C03601=1040.712,-116.263,-73.766,168.679,35.382,156.678
C03602=1040.719,-115.977,-73.778,168.682,35.382,156.678
C03603=1040.726,-115.691,-73.788,168.684,35.381,156.678
C03604=1040.733,-115.404,-73.799,168.687,35.381,156.678
C03605=1040.739,-115.155,-73.808,168.690,35.381,156.678
C03606=1040.745,-114.905,-73.817,168.692,35.380,156.678
C03607=1040.751,-114.656,-73.827,168.695,35.380,156.678
C03608=1040.757,-114.406,-73.837,168.698,35.380,156.678
C03609=1040.763,-114.156,-73.846,168.700,35.379,156.678
C03610=1040.769,-113.906,-73.855,168.703,35.378,156.677
C03611=1040.775,-113.656,-73.865,168.705,35.379,156.677
C03612=1040.781,-113.406,-73.874,168.708,35.378,156.677
C03613=1040.787,-113.157,-73.883,168.710,35.378,156.677
C03614=1040.793,-112.907,-73.893,168.712,35.377,156.677
C03615=1040.799,-112.657,-73.902,168.714,35.377,156.677
C03616=1040.806,-112.407,-73.912,168.717,35.377,156.677
C03617=1040.812,-112.158,-73.922,168.719,35.376,156.677
C03618=1040.818,-111.908,-73.931,168.722,35.376,156.677
C03619=1040.823,-111.658,-73.941,168.724,35.376,156.677
C03620=1040.829,-111.408,-73.951,168.727,35.375,156.677
C03621=1040.836,-111.158,-73.960,168.729,35.375,156.677
C03622=1040.841,-110.909,-73.970,168.732,35.375,156.676
C03623=1040.847,-110.659,-73.979,168.734,35.375,156.676
C03624=1040.854,-110.409,-73.989,168.737,35.374,156.676
C03625=1040.860,-110.160,-73.999,168.740,35.374,156.676
C03626=1040.866,-109.911,-74.009,168.742,35.374,156.676
C03627=1040.872,-109.661,-74.018,168.745,35.373,156.676
C03628=1040.879,-109.411,-74.028,168.747,35.373,156.676
C03629=1040.885,-109.161,-74.037,168.750,35.373,156.676
C03630=1040.891,-108.911,-74.047,168.752,35.373,156.676
C03631=1040.897,-108.662,-74.056,168.755,35.372,156.676
C03632=1040.903,-108.412,-74.066,168.757,35.372,156.676
C03633=1040.909,-108.162,-74.076,168.760,35.372,156.676
C03634=1040.915,-107.912,-74.086,168.762,35.372,156.676
C03635=1040.921,-107.663,-74.096,168.765,35.371,156.675
C03636=1040.927,-107.413,-74.106,168.767,35.371,156.675
C03637=1040.934,-107.163,-74.115,168.770,35.371,156.675
C03638=1040.940,-106.913,-74.125,168.772,35.371,156.675
C03639=1040.945,-106.663,-74.135,168.775,35.370,156.675
C03640=1040.952,-106.414,-74.145,168.777,35.370,156.675
C03641=1040.958,-106.164,-74.155,168.779,35.370,156.675
C03642=1040.964,-105.914,-74.164,168.781,35.370,156.675
C03643=1040.970,-105.665,-74.174,168.784,35.370,156.675
C03644=1040.976,-105.414,-74.184,168.786,35.369,156.675
C03645=1040.982,-105.165,-74.194,168.789,35.369,156.675
C03646=1040.988,-104.915,-74.204,168.791,35.369,156.675
C03647=1040.994,-104.666,-74.213,168.794,35.369,156.675
C03648=1041.000,-104.416,-74.224,168.796,35.369,156.675
C03649=1041.006,-104.166,-74.234,168.799,35.368,156.674
C03650=1041.013,-103.917,-74.243,168.801,35.368,156.674
C03651=1041.019,-103.667,-74.253,168.804,35.368,156.674
C03652=1041.024,-103.417,-74.264,168.806,35.368,156.674
C03653=1041.031,-103.168,-74.273,168.809,35.368,156.674
C03654=1041.037,-102.918,-74.283,168.811,35.367,156.674
C03655=1041.043,-102.668,-74.294,168.814,35.368,156.674
C03656=1041.049,-102.418,-74.303,168.816,35.368,156.674
C03657=1041.055,-102.169,-74.313,168.819,35.367,156.674
C03658=1041.061,-101.919,-74.323,168.821,35.367,156.674
C03659=1041.067,-101.669,-74.334,168.824,35.367,156.674
C03660=1041.074,-101.419,-74.344,168.826,35.367,156.674
C03661=1041.080,-101.170,-74.354,168.829,35.367,156.674
C03662=1041.086,-100.920,-74.364,168.831,35.367,156.674
C03663=1041.092,-100.670,-74.374,168.834,35.366,156.674
C03664=1041.098,-100.421,-74.384,168.836,35.366,156.674
C03665=1041.105,-100.134,-74.396,168.839,35.366,156.674
C03666=1041.112,-99.846,-74.408,168.842,35.366,156.673
C03667=1041.120,-99.559,-74.419,168.845,35.366,156.673
C03668=1041.127,-99.272,-74.431,168.847,35.366,156.673
C03669=1041.133,-99.022,-74.441,168.850,35.365,156.673
C03670=1041.139,-98.772,-74.450,168.852,35.365,156.673
C03671=1041.145,-98.523,-74.461,168.855,35.366,156.673
C03672=1041.151,-98.273,-74.471,168.857,35.366,156.673
C03673=1041.157,-98.024,-74.481,168.860,35.365,156.673
C03674=1041.163,-97.773,-74.492,168.862,35.365,156.673
C03675=1041.170,-97.524,-74.502,168.865,35.365,156.673
C03676=1041.175,-97.274,-74.512,168.867,35.365,156.673
C03677=1041.182,-97.025,-74.522,168.870,35.365,156.673
C03678=1041.187,-96.775,-74.533,168.871,35.365,156.673
C03679=1041.194,-96.525,-74.543,168.874,35.365,156.673
C03680=1041.199,-96.276,-74.554,168.876,35.365,156.673
C03681=1041.206,-96.025,-74.564,168.878,35.365,156.673
C03682=1041.212,-95.776,-74.575,168.881,35.365,156.673
C03683=1041.218,-95.526,-74.585,168.883,35.365,156.673
C03684=1041.224,-95.277,-74.595,168.886,35.365,156.673
C03685=1041.230,-95.027,-74.606,168.888,35.365,156.673
C03686=1041.236,-94.778,-74.616,168.891,35.365,156.673
C03687=1041.242,-94.527,-74.627,168.893,35.365,156.673
C03688=1041.248,-94.278,-74.637,168.895,35.365,156.673
C03689=1041.254,-94.028,-74.648,168.898,35.366,156.673
C03690=1041.260,-93.778,-74.658,168.900,35.365,156.673
C03691=1041.266,-93.529,-74.668,168.903,35.365,156.673
C03692=1041.272,-93.279,-74.680,168.905,35.365,156.673
C03693=1041.279,-93.029,-74.689,168.908,35.365,156.673
C03694=1041.284,-92.780,-74.700,168.910,35.365,156.673
C03695=1041.290,-92.530,-74.711,168.913,35.365,156.673
C03696=1041.297,-92.280,-74.721,168.915,35.365,156.672
C03697=1041.303,-92.030,-74.732,168.917,35.366,156.672
C03698=1041.309,-91.781,-74.742,168.920,35.366,156.672
C03699=1041.315,-91.531,-74.753,168.922,35.366,156.672
C03700=1041.321,-91.281,-74.764,168.925,35.366,156.672
C03701=1041.327,-91.031,-74.774,168.927,35.366,156.672
C03702=1041.333,-90.782,-74.785,168.930,35.366,156.672
C03703=1041.340,-90.533,-74.795,168.932,35.366,156.672
C03704=1041.346,-90.283,-74.806,168.934,35.366,156.672
C03705=1041.351,-90.033,-74.816,168.937,35.366,156.672
C03706=1041.358,-89.783,-74.826,168.939,35.366,156.672
C03707=1041.364,-89.533,-74.838,168.942,35.366,156.672
C03708=1041.370,-89.284,-74.849,168.944,35.366,156.672
C03709=1041.376,-89.034,-74.859,168.946,35.366,156.672
C03710=1041.382,-88.785,-74.870,168.949,35.366,156.672
C03711=1041.389,-88.535,-74.880,168.951,35.367,156.672
C03712=1041.395,-88.285,-74.891,168.954,35.367,156.672
C03713=1041.400,-88.036,-74.901,168.956,35.367,156.672
C03714=1041.407,-87.786,-74.912,168.959,35.367,156.672
C03715=1041.413,-87.536,-74.923,168.961,35.367,156.672
C03716=1041.419,-87.287,-74.934,168.963,35.367,156.672
C03717=1041.426,-87.037,-74.944,168.966,35.367,156.672
C03718=1041.432,-86.787,-74.955,168.968,35.367,156.672
C03719=1041.438,-86.537,-74.967,168.971,35.367,156.672
C03720=1041.445,-86.288,-74.977,168.973,35.367,156.672
C03721=1041.450,-86.038,-74.988,168.975,35.367,156.672
C03722=1041.456,-85.788,-74.998,168.978,35.367,156.672
C03723=1041.463,-85.538,-75.009,168.980,35.367,156.672
C03724=1041.469,-85.289,-75.019,168.983,35.367,156.672
C03725=1041.475,-85.039,-75.031,168.985,35.368,156.672
C03726=1041.481,-84.790,-75.041,168.988,35.368,156.672
C03727=1041.488,-84.539,-75.052,168.990,35.368,156.672
C03728=1041.493,-84.290,-75.063,168.992,35.368,156.672
C03729=1041.501,-84.005,-75.076,168.995,35.369,156.672
C03730=1041.508,-83.721,-75.088,168.998,35.369,156.672
C03731=1041.515,-83.435,-75.100,169.001,35.369,156.672
C03732=1041.522,-83.151,-75.113,169.003,35.369,156.672
C03733=1041.529,-82.901,-75.124,169.006,35.369,156.672
C03734=1041.535,-82.652,-75.135,169.008,35.369,156.672
C03735=1041.541,-82.402,-75.146,169.011,35.369,156.672
C03736=1041.547,-82.152,-75.157,169.013,35.369,156.672
C03737=1041.554,-81.902,-75.167,169.015,35.369,156.672
C03738=1041.560,-81.653,-75.178,169.018,35.369,156.672
C03739=1041.566,-81.403,-75.189,169.020,35.370,156.672
C03740=1041.573,-81.153,-75.200,169.023,35.370,156.672
C03741=1041.579,-80.903,-75.211,169.025,35.370,156.672
C03742=1041.585,-80.654,-75.222,169.027,35.370,156.672
C03743=1041.591,-80.403,-75.233,169.030,35.370,156.672
C03744=1041.598,-80.155,-75.244,169.032,35.370,156.672
C03745=1041.604,-79.905,-75.255,169.035,35.370,156.672
C03746=1041.610,-79.655,-75.266,169.037,35.370,156.672
C03747=1041.616,-79.405,-75.277,169.039,35.371,156.672
C03748=1041.622,-79.156,-75.288,169.042,35.371,156.672
C03749=1041.628,-78.905,-75.300,169.044,35.371,156.672
C03750=1041.634,-78.656,-75.311,169.046,35.372,156.672
C03751=1041.642,-78.407,-75.322,169.049,35.372,156.672
C03752=1041.647,-78.157,-75.333,169.051,35.372,156.672
C03753=1041.654,-77.907,-75.344,169.053,35.372,156.672
C03754=1041.660,-77.658,-75.356,169.056,35.373,156.672
C03755=1041.666,-77.408,-75.367,169.058,35.373,156.672
C03756=1041.672,-77.158,-75.378,169.060,35.373,156.672
C03757=1041.678,-76.909,-75.390,169.063,35.374,156.672
C03758=1041.684,-76.659,-75.400,169.065,35.374,156.672
C03759=1041.690,-76.409,-75.412,169.068,35.374,156.672
C03760=1041.696,-76.160,-75.423,169.070,35.375,156.672
C03761=1041.703,-75.910,-75.435,169.072,35.375,156.672
C03762=1041.709,-75.661,-75.445,169.075,35.375,156.672
C03763=1041.715,-75.410,-75.457,169.077,35.375,156.672
C03764=1041.722,-75.161,-75.469,169.079,35.376,156.672
C03765=1041.727,-74.911,-75.480,169.082,35.376,156.672
C03766=1041.734,-74.661,-75.491,169.084,35.376,156.672
C03767=1041.740,-74.412,-75.502,169.086,35.376,156.672
C03768=1041.746,-74.162,-75.514,169.089,35.376,156.672
C03769=1041.752,-73.913,-75.525,169.091,35.377,156.672
C03770=1041.758,-73.663,-75.536,169.093,35.377,156.672
C03771=1041.765,-73.413,-75.548,169.096,35.378,156.672
C03772=1041.771,-73.164,-75.559,169.098,35.378,156.672
C03773=1041.776,-72.913,-75.571,169.100,35.379,156.673
C03774=1041.782,-72.665,-75.583,169.103,35.379,156.672
C03775=1041.789,-72.414,-75.594,169.105,35.380,156.673
C03776=1041.795,-72.166,-75.606,169.107,35.380,156.673
C03777=1041.800,-71.915,-75.617,169.109,35.380,156.673
C03778=1041.807,-71.665,-75.629,169.112,35.380,156.673
C03779=1041.813,-71.416,-75.640,169.114,35.381,156.673
C03780=1041.820,-71.166,-75.652,169.116,35.381,156.673
C03781=1041.825,-70.917,-75.664,169.119,35.382,156.673
C03782=1041.831,-70.667,-75.676,169.121,35.382,156.673
C03783=1041.837,-70.417,-75.687,169.123,35.383,156.673
C03784=1041.844,-70.168,-75.698,169.126,35.383,156.673
C03785=1041.850,-69.918,-75.710,169.128,35.383,156.673
C03786=1041.855,-69.669,-75.722,169.130,35.384,156.673
C03787=1041.862,-69.419,-75.734,169.132,35.384,156.673
C03788=1041.868,-69.169,-75.745,169.135,35.385,156.673
C03789=1041.874,-68.920,-75.757,169.137,35.385,156.673
C03790=1041.880,-68.669,-75.768,169.139,35.386,156.673
C03791=1041.886,-68.420,-75.780,169.142,35.386,156.673
C03792=1041.893,-68.171,-75.792,169.144,35.386,156.673
C03793=1041.899,-67.888,-75.805,169.147,35.387,156.673
C03794=1041.907,-67.605,-75.818,169.149,35.387,156.673
C03795=1041.914,-67.323,-75.832,169.152,35.388,156.673
C03796=1041.920,-67.040,-75.845,169.154,35.389,156.674
C03797=1041.926,-66.790,-75.857,169.157,35.389,156.674
C03798=1041.933,-66.540,-75.869,169.159,35.390,156.674
C03799=1041.939,-66.291,-75.881,169.161,35.390,156.674
C03800=1041.945,-66.042,-75.892,169.163,35.390,156.674
C03801=1041.951,-65.791,-75.904,169.166,35.390,156.674
C03802=1041.957,-65.542,-75.916,169.168,35.391,156.674
C03803=1041.964,-65.293,-75.928,169.170,35.392,156.674
C03804=1041.969,-65.042,-75.940,169.173,35.392,156.674
C03805=1041.976,-64.793,-75.952,169.175,35.393,156.674
C03806=1041.982,-64.544,-75.963,169.177,35.393,156.674
C03807=1041.989,-64.294,-75.975,169.179,35.393,156.674
C03808=1041.994,-64.044,-75.987,169.182,35.394,156.674
C03809=1042.001,-63.794,-75.999,169.184,35.394,156.674
C03810=1042.007,-63.545,-76.011,169.186,35.395,156.674
C03811=1042.013,-63.295,-76.023,169.189,35.395,156.674
C03812=1042.019,-63.045,-76.034,169.192,35.396,156.674
C03813=1042.026,-62.796,-76.046,169.194,35.396,156.674
C03814=1042.031,-62.546,-76.059,169.196,35.396,156.674
C03815=1042.038,-62.297,-76.071,169.199,35.397,156.675
C03816=1042.044,-62.047,-76.082,169.201,35.398,156.675
C03817=1042.050,-61.797,-76.095,169.203,35.398,156.675
C03818=1042.057,-61.547,-76.106,169.205,35.399,156.675
C03819=1042.063,-61.298,-76.118,169.208,35.399,156.675
C03820=1042.069,-61.049,-76.130,169.210,35.399,156.675
C03821=1042.075,-60.799,-76.142,169.212,35.400,156.675
C03822=1042.082,-60.549,-76.154,169.214,35.400,156.675
C03823=1042.088,-60.300,-76.166,169.217,35.401,156.675
C03824=1042.094,-60.050,-76.179,169.219,35.402,156.675
C03825=1042.100,-59.800,-76.190,169.221,35.402,156.675
C03826=1042.107,-59.551,-76.202,169.224,35.402,156.675
C03827=1042.113,-59.301,-76.214,169.226,35.403,156.675
C03828=1042.119,-59.051,-76.226,169.228,35.403,156.675
C03829=1042.126,-58.802,-76.238,169.230,35.404,156.675
C03830=1042.132,-58.552,-76.251,169.233,35.405,156.675
C03831=1042.139,-58.302,-76.263,169.235,35.405,156.675
C03832=1042.144,-58.053,-76.275,169.237,35.405,156.675
C03833=1042.150,-57.804,-76.287,169.239,35.406,156.676
C03834=1042.157,-57.554,-76.299,169.242,35.406,156.676
C03835=1042.163,-57.304,-76.311,169.244,35.407,156.676
C03836=1042.170,-57.055,-76.323,169.246,35.407,156.676
C03837=1042.176,-56.805,-76.335,169.248,35.408,156.676
C03838=1042.182,-56.555,-76.348,169.251,35.408,156.676
C03839=1042.189,-56.306,-76.360,169.253,35.409,156.676
C03840=1042.196,-56.056,-76.372,169.255,35.409,156.676
C03841=1042.201,-55.806,-76.384,169.257,35.410,156.676
C03842=1042.208,-55.556,-76.396,169.260,35.410,156.676
C03843=1042.214,-55.308,-76.408,169.262,35.410,156.676
C03844=1042.220,-55.058,-76.420,169.264,35.411,156.676
C03845=1042.227,-54.808,-76.432,169.266,35.412,156.676
C03846=1042.233,-54.558,-76.445,169.269,35.412,156.676
C03847=1042.239,-54.309,-76.457,169.271,35.413,156.676
C03848=1042.246,-54.059,-76.469,169.273,35.413,156.676
C03849=1042.252,-53.809,-76.481,169.275,35.414,156.677
C03850=1042.259,-53.560,-76.494,169.278,35.414,156.677
C03851=1042.265,-53.310,-76.507,169.280,35.415,156.677
C03852=1042.271,-53.061,-76.519,169.282,35.416,156.677
C03853=1042.278,-52.811,-76.531,169.284,35.416,156.677
C03854=1042.284,-52.561,-76.543,169.286,35.416,156.677
C03855=1042.291,-52.312,-76.555,169.289,35.417,156.677
C03856=1042.296,-52.062,-76.568,169.291,35.417,156.677
C03857=1042.305,-51.781,-76.581,169.293,35.418,156.677
C03858=1042.312,-51.499,-76.596,169.297,35.419,156.677
C03859=1042.318,-51.218,-76.609,169.299,35.419,156.677
C03860=1042.326,-50.937,-76.624,169.302,35.420,156.677
C03861=1042.332,-50.687,-76.636,169.304,35.420,156.677
C03862=1042.338,-50.437,-76.648,169.306,35.421,156.677
C03863=1042.345,-50.188,-76.660,169.309,35.421,156.677
C03864=1042.351,-49.938,-76.673,169.311,35.422,156.678
C03865=1042.357,-49.688,-76.686,169.313,35.423,156.678
C03866=1042.364,-49.439,-76.698,169.315,35.424,156.678
C03867=1042.370,-49.189,-76.710,169.317,35.424,156.678
C03868=1042.376,-48.940,-76.724,169.319,35.425,156.678
C03869=1042.382,-48.690,-76.736,169.322,35.426,156.678
C03870=1042.388,-48.440,-76.748,169.324,35.426,156.678
C03871=1042.395,-48.191,-76.761,169.326,35.427,156.678
C03872=1042.400,-47.941,-76.774,169.328,35.428,156.678
C03873=1042.407,-47.692,-76.787,169.330,35.428,156.678
C03874=1042.413,-47.442,-76.799,169.333,35.429,156.679
C03875=1042.419,-47.192,-76.812,169.335,35.430,156.679
C03876=1042.425,-46.943,-76.825,169.337,35.431,156.679
C03877=1042.431,-46.693,-76.838,169.339,35.431,156.679
C03878=1042.438,-46.444,-76.850,169.341,35.432,156.679
C03879=1042.445,-46.194,-76.863,169.343,35.433,156.679
C03880=1042.451,-45.944,-76.876,169.346,35.433,156.679
C03881=1042.457,-45.695,-76.889,169.348,35.434,156.679
C03882=1042.463,-45.445,-76.902,169.350,35.435,156.679
C03883=1042.469,-45.195,-76.914,169.352,35.435,156.679
C03884=1042.476,-44.946,-76.927,169.354,35.436,156.679
C03885=1042.482,-44.696,-76.939,169.356,35.436,156.680
C03886=1042.488,-44.447,-76.953,169.359,35.437,156.680
C03887=1042.494,-44.197,-76.965,169.362,35.438,156.680
C03888=1042.501,-43.948,-76.978,169.364,35.438,156.680
C03889=1042.507,-43.698,-76.990,169.366,35.439,156.680
C03890=1042.513,-43.449,-77.004,169.368,35.440,156.680
C03891=1042.519,-43.198,-77.017,169.370,35.440,156.680
C03892=1042.526,-42.949,-77.029,169.372,35.441,156.680
C03893=1042.532,-42.699,-77.042,169.375,35.442,156.680
C03894=1042.538,-42.450,-77.055,169.377,35.443,156.680
C03895=1042.544,-42.200,-77.068,169.379,35.443,156.681
C03896=1042.551,-41.951,-77.080,169.381,35.444,156.681
C03897=1042.557,-41.701,-77.093,169.383,35.445,156.681
C03898=1042.564,-41.451,-77.107,169.385,35.445,156.681
C03899=1042.570,-41.202,-77.120,169.387,35.446,156.681
C03900=1042.576,-40.952,-77.132,169.390,35.447,156.681
C03901=1042.582,-40.703,-77.146,169.392,35.447,156.681
C03902=1042.589,-40.453,-77.158,169.394,35.448,156.681
C03903=1042.595,-40.204,-77.171,169.396,35.449,156.681
C03904=1042.602,-39.954,-77.185,169.398,35.450,156.682
C03905=1042.608,-39.704,-77.197,169.400,35.451,156.682
C03906=1042.614,-39.455,-77.210,169.402,35.452,156.682
C03907=1042.621,-39.205,-77.222,169.405,35.452,156.682
C03908=1042.627,-38.956,-77.236,169.407,35.453,156.682
C03909=1042.634,-38.706,-77.249,169.409,35.454,156.682
C03910=1042.640,-38.456,-77.262,169.411,35.454,156.682
C03911=1042.646,-38.207,-77.275,169.414,35.455,156.682
C03912=1042.652,-37.958,-77.288,169.416,35.456,156.682
C03913=1042.658,-37.708,-77.301,169.418,35.456,156.682
C03914=1042.665,-37.458,-77.314,169.420,35.458,156.683
C03915=1042.671,-37.209,-77.328,169.423,35.459,156.683
C03916=1042.677,-36.959,-77.341,169.425,35.459,156.683
C03917=1042.683,-36.710,-77.354,169.427,35.460,156.683
C03918=1042.689,-36.460,-77.367,169.429,35.461,156.683
C03919=1042.695,-36.210,-77.381,169.431,35.461,156.683
C03920=1042.702,-35.961,-77.394,169.433,35.463,156.683
C03921=1042.708,-35.680,-77.408,169.435,35.463,156.683
C03922=1042.716,-35.399,-77.424,169.438,35.464,156.684
C03923=1042.723,-35.118,-77.439,169.440,35.465,156.684
C03924=1042.730,-34.837,-77.453,169.442,35.466,156.684
C03925=1042.737,-34.587,-77.467,169.445,35.467,156.684
C03926=1042.743,-34.338,-77.480,169.447,35.467,156.684
C03927=1042.749,-34.088,-77.493,169.449,35.469,156.684
C03928=1042.755,-33.839,-77.506,169.451,35.469,156.684
C03929=1042.762,-33.589,-77.520,169.453,35.470,156.684
C03930=1042.767,-33.340,-77.534,169.455,35.471,156.685
C03931=1042.773,-33.090,-77.547,169.458,35.472,156.685
C03932=1042.780,-32.840,-77.560,169.460,35.473,156.685
C03933=1042.786,-32.591,-77.574,169.462,35.474,156.685
C03934=1042.792,-32.341,-77.586,169.464,35.474,156.685
C03935=1042.799,-32.092,-77.600,169.466,35.475,156.685
C03936=1042.805,-31.842,-77.613,169.469,35.476,156.685
C03937=1042.812,-31.593,-77.626,169.471,35.477,156.686
C03938=1042.818,-31.343,-77.640,169.473,35.478,156.686
C03939=1042.825,-31.093,-77.653,169.475,35.478,156.686
C03940=1042.831,-30.844,-77.667,169.477,35.479,156.686
C03941=1042.836,-30.595,-77.681,169.479,35.480,156.686
C03942=1042.843,-30.345,-77.694,169.481,35.481,156.686
C03943=1042.849,-30.095,-77.707,169.483,35.482,156.686
C03944=1042.856,-29.846,-77.721,169.485,35.483,156.686
C03945=1042.862,-29.596,-77.734,169.487,35.483,156.686
C03946=1042.869,-29.347,-77.748,169.489,35.484,156.687
C03947=1042.875,-29.098,-77.761,169.491,35.485,156.687
C03948=1042.882,-28.848,-77.775,169.493,35.486,156.687
C03949=1042.888,-28.598,-77.788,169.495,35.487,156.687
C03950=1042.894,-28.348,-77.802,169.498,35.487,156.687
C03951=1042.900,-28.099,-77.815,169.501,35.489,156.687
C03952=1042.906,-27.850,-77.829,169.503,35.489,156.687
C03953=1042.913,-27.600,-77.842,169.505,35.490,156.687
C03954=1042.919,-27.350,-77.855,169.507,35.491,156.688
C03955=1042.926,-27.100,-77.869,169.509,35.491,156.688
C03956=1042.932,-26.851,-77.882,169.511,35.493,156.688
C03957=1042.938,-26.602,-77.896,169.513,35.493,156.688
C03958=1042.945,-26.352,-77.910,169.515,35.494,156.688
C03959=1042.951,-26.102,-77.923,169.517,35.495,156.688
C03960=1042.957,-25.853,-77.938,169.519,35.496,156.688
C03961=1042.964,-25.603,-77.951,169.521,35.497,156.689
C03962=1042.969,-25.354,-77.965,169.523,35.498,156.689
C03963=1042.976,-25.104,-77.979,169.525,35.499,156.689
C03964=1042.982,-24.855,-77.992,169.527,35.500,156.689
C03965=1042.988,-24.605,-78.006,169.529,35.501,156.689
C03966=1042.995,-24.356,-78.020,169.531,35.502,156.689
C03967=1043.001,-24.106,-78.034,169.533,35.503,156.689
C03968=1043.007,-23.856,-78.048,169.536,35.504,156.690
C03969=1043.013,-23.607,-78.061,169.538,35.505,156.690
C03970=1043.019,-23.358,-78.074,169.540,35.506,156.690
C03971=1043.026,-23.108,-78.089,169.542,35.506,156.690
C03972=1043.032,-22.859,-78.103,169.544,35.508,156.690
C03973=1043.038,-22.608,-78.117,169.546,35.508,156.690
C03974=1043.044,-22.359,-78.130,169.548,35.510,156.691
C03975=1043.051,-22.110,-78.144,169.550,35.510,156.691
C03976=1043.057,-21.860,-78.158,169.552,35.511,156.691
C03977=1043.064,-21.610,-78.172,169.554,35.512,156.691
C03978=1043.069,-21.361,-78.186,169.556,35.513,156.691
C03979=1043.076,-21.112,-78.200,169.558,35.514,156.691
C03980=1043.082,-20.862,-78.213,169.560,35.515,156.691
C03981=1043.088,-20.612,-78.227,169.562,35.516,156.691
C03982=1043.095,-20.363,-78.242,169.564,35.517,156.692
C03983=1043.101,-20.114,-78.255,169.566,35.518,156.692
C03984=1043.107,-19.864,-78.269,169.569,35.519,156.692
C03985=1043.115,-19.582,-78.285,169.572,35.520,156.692
C03986=1043.122,-19.301,-78.301,169.574,35.521,156.692
C03987=1043.129,-19.018,-78.316,169.576,35.522,156.692
C03988=1043.136,-18.737,-78.332,169.579,35.523,156.693
C03989=1043.142,-18.487,-78.346,169.581,35.524,156.693
C03990=1043.149,-18.238,-78.360,169.583,35.525,156.693
C03991=1043.155,-17.988,-78.374,169.585,35.526,156.693
C03992=1043.162,-17.739,-78.389,169.586,35.527,156.693
C03993=1043.168,-17.489,-78.402,169.588,35.528,156.693
C03994=1043.174,-17.239,-78.416,169.590,35.529,156.693
C03995=1043.181,-16.990,-78.430,169.592,35.530,156.694
C03996=1043.187,-16.740,-78.444,169.594,35.531,156.694
C03997=1043.193,-16.491,-78.459,169.596,35.531,156.694
C03998=1043.200,-16.241,-78.472,169.598,35.533,156.694
C03999=1043.206,-15.993,-78.487,169.600,35.533,156.694
C04000=1043.213,-15.743,-78.500,169.603,35.535,156.694
C04001=1043.219,-15.492,-78.515,169.605,35.535,156.695
C04002=1043.225,-15.244,-78.529,169.607,35.536,156.695
C04003=1043.231,-14.993,-78.543,169.609,35.537,156.695
C04004=1043.238,-14.745,-78.557,169.611,35.539,156.695
C04005=1043.244,-14.495,-78.572,169.613,35.539,156.695
C04006=1043.250,-14.245,-78.586,169.615,35.541,156.695
C04007=1043.257,-13.996,-78.600,169.617,35.541,156.695
C04008=1043.263,-13.746,-78.614,169.619,35.543,156.696
C04009=1043.269,-13.497,-78.629,169.621,35.543,156.696
C04010=1043.275,-13.247,-78.642,169.623,35.545,156.696
C04011=1043.281,-12.998,-78.657,169.625,35.545,156.696
C04012=1043.288,-12.748,-78.672,169.627,35.547,156.696
C04013=1043.294,-12.498,-78.686,169.629,35.548,156.697
C04014=1043.300,-12.249,-78.700,169.631,35.549,156.697
C04015=1043.306,-11.999,-78.714,169.634,35.550,156.697
C04016=1043.313,-11.750,-78.728,169.636,35.551,156.697
C04017=1043.319,-11.501,-78.743,169.638,35.552,156.697
C04018=1043.325,-11.251,-78.758,169.640,35.553,156.697
C04019=1043.332,-11.002,-78.772,169.642,35.554,156.698
C04020=1043.338,-10.752,-78.787,169.644,35.555,156.698
C04021=1043.344,-10.503,-78.800,169.646,35.556,156.698
C04022=1043.351,-10.253,-78.815,169.647,35.557,156.698
C04023=1043.357,-10.004,-78.830,169.649,35.558,156.698
C04024=1043.363,-9.754,-78.844,169.651,35.559,156.698
C04025=1043.369,-9.504,-78.859,169.653,35.560,156.698
C04026=1043.376,-9.255,-78.873,169.655,35.561,156.699
C04027=1043.382,-9.006,-78.887,169.657,35.562,156.699
C04028=1043.388,-8.756,-78.902,169.660,35.563,156.699
C04029=1043.395,-8.507,-78.916,169.662,35.564,156.699
C04030=1043.401,-8.258,-78.931,169.664,35.565,156.699
C04031=1043.407,-8.007,-78.945,169.666,35.567,156.700
C04032=1043.414,-7.758,-78.959,169.668,35.567,156.700
C04033=1043.420,-7.509,-78.974,169.670,35.569,156.700
C04034=1043.426,-7.259,-78.989,169.672,35.569,156.700
C04035=1043.432,-7.009,-79.003,169.674,35.571,156.700
C04036=1043.439,-6.760,-79.017,169.676,35.571,156.700
C04037=1043.445,-6.511,-79.032,169.678,35.573,156.701
C04038=1043.452,-6.261,-79.047,169.679,35.574,156.701
C04039=1043.459,-6.012,-79.061,169.681,35.575,156.701
C04040=1043.464,-5.762,-79.075,169.683,35.576,156.701
C04041=1043.471,-5.513,-79.090,169.685,35.577,156.701
C04042=1043.477,-5.263,-79.105,169.688,35.578,156.701
C04043=1043.484,-5.014,-79.119,169.690,35.579,156.701
C04044=1043.490,-4.765,-79.134,169.692,35.580,156.702
C04045=1043.496,-4.515,-79.149,169.694,35.581,156.702
C04046=1043.502,-4.265,-79.163,169.696,35.582,156.702
C04047=1043.509,-4.015,-79.177,169.698,35.583,156.702
C04048=1043.515,-3.766,-79.192,169.700,35.584,156.702
C04049=1043.523,-3.483,-79.209,169.702,35.585,156.703
C04050=1043.530,-3.199,-79.226,169.704,35.587,156.703
C04051=1043.537,-2.915,-79.243,169.706,35.588,156.703
C04052=1043.544,-2.633,-79.260,169.708,35.589,156.703
C04053=1043.550,-2.384,-79.274,169.710,35.590,156.703
C04054=1043.556,-2.134,-79.289,169.712,35.591,156.704
C04055=1043.563,-1.884,-79.304,169.715,35.592,156.704
C04056=1043.569,-1.635,-79.319,169.717,35.594,156.704
C04057=1043.575,-1.386,-79.334,169.719,35.595,156.704
C04058=1043.581,-1.136,-79.349,169.721,35.596,156.704
C04059=1043.587,-0.886,-79.364,169.722,35.597,156.705
C04060=1043.594,-0.637,-79.379,169.724,35.598,156.705
C04061=1043.600,-0.388,-79.393,169.726,35.600,156.705
C04062=1043.606,-0.138,-79.408,169.728,35.600,156.705
C04063=1043.612,0.111,-79.423,169.730,35.602,156.705
C04064=1043.619,0.361,-79.438,169.732,35.603,156.706
C04065=1043.624,0.610,-79.453,169.734,35.604,156.706
C04066=1043.630,0.860,-79.468,169.736,35.605,156.706
C04067=1043.637,1.110,-79.483,169.738,35.606,156.706
C04068=1043.643,1.359,-79.498,169.740,35.608,156.706
C04069=1043.649,1.609,-79.513,169.742,35.609,156.706
C04070=1043.655,1.858,-79.528,169.744,35.610,156.707
C04071=1043.662,2.107,-79.543,169.746,35.611,156.707
C04072=1043.668,2.357,-79.558,169.748,35.612,156.707
C04073=1043.675,2.606,-79.573,169.750,35.614,156.707
C04074=1043.681,2.856,-79.588,169.751,35.614,156.707
C04075=1043.687,3.106,-79.603,169.753,35.616,156.708
C04076=1043.693,3.355,-79.618,169.755,35.617,156.708
C04077=1043.700,3.604,-79.633,169.757,35.618,156.708
C04078=1043.706,3.853,-79.648,169.760,35.619,156.708
C04079=1043.713,4.103,-79.663,169.762,35.620,156.708
C04080=1043.718,4.353,-79.679,169.764,35.621,156.709
C04081=1043.725,4.603,-79.694,169.765,35.623,156.709
C04082=1043.731,4.852,-79.709,169.767,35.623,156.709
C04083=1043.737,5.101,-79.724,169.769,35.625,156.709
C04084=1043.744,5.350,-79.739,169.771,35.626,156.709
C04085=1043.750,5.600,-79.754,169.773,35.627,156.710
C04086=1043.756,5.850,-79.769,169.775,35.628,156.710
C04087=1043.763,6.099,-79.784,169.777,35.629,156.710
C04088=1043.769,6.348,-79.799,169.778,35.631,156.710
C04089=1043.776,6.598,-79.814,169.780,35.632,156.710
C04090=1043.781,6.848,-79.830,169.783,35.633,156.710
C04091=1043.788,7.098,-79.845,169.785,35.634,156.711
C04092=1043.794,7.346,-79.860,169.787,35.635,156.711
C04093=1043.800,7.596,-79.875,169.789,35.637,156.711
C04094=1043.807,7.845,-79.890,169.791,35.637,156.711
C04095=1043.813,8.094,-79.906,169.792,35.639,156.711
C04096=1043.820,8.344,-79.921,169.794,35.640,156.712
C04097=1043.826,8.594,-79.936,169.796,35.641,156.712
C04098=1043.833,8.843,-79.951,169.798,35.642,156.712
C04099=1043.838,9.093,-79.967,169.800,35.643,156.712
C04100=1043.845,9.342,-79.982,169.802,35.644,156.712
C04101=1043.851,9.591,-79.997,169.804,35.646,156.713
C04102=1043.858,9.841,-80.012,169.806,35.646,156.713
C04103=1043.864,10.091,-80.027,169.808,35.648,156.713
C04104=1043.871,10.340,-80.043,169.810,35.649,156.713
C04105=1043.877,10.589,-80.058,169.812,35.650,156.713
C04106=1043.884,10.839,-80.073,169.814,35.651,156.714
C04107=1043.890,11.088,-80.089,169.816,35.652,156.714
C04108=1043.896,11.338,-80.104,169.817,35.654,156.714
C04109=1043.903,11.587,-80.120,169.819,35.655,156.714
C04110=1043.909,11.837,-80.135,169.821,35.656,156.714
C04111=1043.915,12.086,-80.150,169.823,35.657,156.714
C04112=1043.922,12.335,-80.165,169.825,35.658,156.715
C04113=1043.930,12.620,-80.183,169.828,35.660,156.715
C04114=1043.937,12.906,-80.200,169.830,35.661,156.715
C04115=1043.944,13.191,-80.217,169.832,35.662,156.715
C04116=1043.951,13.476,-80.235,169.834,35.663,156.716
C04117=1043.957,13.725,-80.251,169.836,35.664,156.716
C04118=1043.964,13.975,-80.266,169.838,35.665,156.716
C04119=1043.970,14.224,-80.282,169.840,35.667,156.716
C04120=1043.976,14.474,-80.297,169.841,35.668,156.716
C04121=1043.983,14.723,-80.313,169.843,35.669,156.717
C04122=1043.989,14.973,-80.328,169.845,35.671,156.717
C04123=1043.995,15.222,-80.344,169.848,35.672,156.717
C04124=1044.001,15.472,-80.359,169.850,35.673,156.717
C04125=1044.008,15.721,-80.375,169.851,35.674,156.717
C04126=1044.014,15.971,-80.391,169.853,35.675,156.718
C04127=1044.021,16.221,-80.406,169.855,35.677,156.718
C04128=1044.027,16.470,-80.423,169.857,35.678,156.718
C04129=1044.033,16.720,-80.437,169.859,35.679,156.718
C04130=1044.040,16.969,-80.453,169.860,35.680,156.718
C04131=1044.046,17.219,-80.469,169.862,35.682,156.719
C04132=1044.052,17.468,-80.484,169.864,35.682,156.719
C04133=1044.058,17.717,-80.501,169.866,35.684,156.719
C04134=1044.065,17.967,-80.516,169.869,35.685,156.719
C04135=1044.072,18.216,-80.531,169.870,35.686,156.719
C04136=1044.077,18.465,-80.547,169.872,35.688,156.720
C04137=1044.084,18.715,-80.562,169.874,35.689,156.720
C04138=1044.090,18.964,-80.579,169.876,35.690,156.720
C04139=1044.096,19.213,-80.594,169.878,35.691,156.720
C04140=1044.103,19.463,-80.609,169.879,35.692,156.720
C04141=1044.109,19.712,-80.626,169.881,35.694,156.721
C04142=1044.116,19.962,-80.642,169.883,35.695,156.721
C04143=1044.122,20.211,-80.658,169.885,35.696,156.721
C04144=1044.128,20.461,-80.673,169.887,35.697,156.721
C04145=1044.134,20.710,-80.689,169.889,35.699,156.722
C04146=1044.141,20.959,-80.705,169.891,35.700,156.722
C04147=1044.147,21.208,-80.721,169.893,35.701,156.722
C04148=1044.153,21.458,-80.736,169.895,35.703,156.722
C04149=1044.159,21.707,-80.752,169.896,35.704,156.722
C04150=1044.165,21.957,-80.768,169.898,35.705,156.723
C04151=1044.172,22.206,-80.784,169.900,35.706,156.723
C04152=1044.178,22.457,-80.800,169.902,35.707,156.723
C04153=1044.185,22.706,-80.816,169.904,35.708,156.723
C04154=1044.191,22.955,-80.832,169.905,35.710,156.723
C04155=1044.198,23.204,-80.848,169.908,35.711,156.724
C04156=1044.204,23.453,-80.864,169.910,35.712,156.724
C04157=1044.209,23.703,-80.880,169.912,35.714,156.724
C04158=1044.216,23.952,-80.895,169.913,35.715,156.724
C04159=1044.222,24.202,-80.911,169.915,35.716,156.725
C04160=1044.229,24.451,-80.927,169.917,35.718,156.725
C04161=1044.235,24.701,-80.944,169.919,35.719,156.725
C04162=1044.242,24.950,-80.959,169.920,35.720,156.725
C04163=1044.248,25.199,-80.975,169.922,35.721,156.725
C04164=1044.254,25.448,-80.992,169.924,35.723,156.726
C04165=1044.260,25.698,-81.007,169.927,35.723,156.726
C04166=1044.267,25.948,-81.023,169.929,35.725,156.726
C04167=1044.273,26.197,-81.039,169.930,35.726,156.726
C04168=1044.279,26.447,-81.055,169.932,35.727,156.726
C04169=1044.286,26.696,-81.071,169.934,35.729,156.727
C04170=1044.292,26.945,-81.087,169.936,35.730,156.727
C04171=1044.298,27.195,-81.104,169.937,35.731,156.727
C04172=1044.305,27.444,-81.119,169.939,35.732,156.727
C04173=1044.311,27.693,-81.136,169.941,35.734,156.728
C04174=1044.317,27.943,-81.152,169.943,35.735,156.728
C04175=1044.324,28.192,-81.168,169.945,35.736,156.728
C04176=1044.330,28.442,-81.184,169.947,35.738,156.728
C04177=1044.338,28.728,-81.203,169.949,35.739,156.729
C04178=1044.345,29.015,-81.221,169.951,35.741,156.729
C04179=1044.351,29.302,-81.240,169.953,35.742,156.729
C04180=1044.359,29.588,-81.259,169.955,35.744,156.729
C04181=1044.365,29.837,-81.275,169.957,35.745,156.730
C04182=1044.371,30.086,-81.291,169.959,35.746,156.730
C04183=1044.378,30.336,-81.307,169.960,35.747,156.730
C04184=1044.384,30.586,-81.323,169.963,35.749,156.730
C04185=1044.390,30.835,-81.340,169.965,35.750,156.730
C04186=1044.396,31.084,-81.356,169.967,35.751,156.731
C04187=1044.402,31.334,-81.373,169.968,35.753,156.731
C04188=1044.409,31.583,-81.389,169.970,35.754,156.731
C04189=1044.415,31.832,-81.405,169.972,35.755,156.731
C04190=1044.421,32.081,-81.421,169.973,35.756,156.732
C04191=1044.428,32.331,-81.438,169.975,35.758,156.732
C04192=1044.434,32.581,-81.454,169.977,35.759,156.732
C04193=1044.440,32.830,-81.470,169.980,35.760,156.732
C04194=1044.446,33.079,-81.486,169.981,35.762,156.732
C04195=1044.453,33.329,-81.504,169.983,35.764,156.733
C04196=1044.459,33.578,-81.520,169.985,35.765,156.733
C04197=1044.465,33.827,-81.536,169.987,35.766,156.733
C04198=1044.471,34.077,-81.552,169.988,35.767,156.733
C04199=1044.478,34.326,-81.568,169.990,35.769,156.734
C04200=1044.484,34.576,-81.585,169.992,35.770,156.734
C04201=1044.491,34.824,-81.602,169.994,35.771,156.734
C04202=1044.497,35.075,-81.618,169.996,35.773,156.734
C04203=1044.503,35.324,-81.635,169.998,35.774,156.735
C04204=1044.509,35.573,-81.651,170.000,35.775,156.735
C04205=1044.517,35.822,-81.668,170.002,35.776,156.735
C04206=1044.523,36.072,-81.684,170.003,35.778,156.735
C04207=1044.529,36.321,-81.700,170.005,35.779,156.735
C04208=1044.535,36.571,-81.717,170.007,35.780,156.736
C04209=1044.541,36.820,-81.734,170.008,35.782,156.736
C04210=1044.547,37.069,-81.750,170.010,35.783,156.736
C04211=1044.555,37.319,-81.766,170.013,35.784,156.736
C04212=1044.561,37.568,-81.782,170.015,35.786,156.737
C04213=1044.567,37.817,-81.799,170.016,35.787,156.737
C04214=1044.573,38.067,-81.816,170.018,35.788,156.737
C04215=1044.580,38.316,-81.833,170.020,35.789,156.737
C04216=1044.586,38.565,-81.849,170.021,35.791,156.738
C04217=1044.592,38.815,-81.866,170.023,35.792,156.738
C04218=1044.598,39.064,-81.883,170.025,35.793,156.738
C04219=1044.604,39.314,-81.899,170.027,35.795,156.738
C04220=1044.610,39.564,-81.916,170.029,35.796,156.739
C04221=1044.616,39.812,-81.933,170.031,35.798,156.739
C04222=1044.622,40.062,-81.949,170.033,35.799,156.739
C04223=1044.629,40.311,-81.967,170.034,35.800,156.739
C04224=1044.635,40.560,-81.983,170.036,35.802,156.739
C04225=1044.641,40.810,-81.999,170.038,35.803,156.740
C04226=1044.648,41.059,-82.016,170.040,35.804,156.740
C04227=1044.654,41.309,-82.033,170.041,35.805,156.740
C04228=1044.661,41.558,-82.050,170.043,35.807,156.740
C04229=1044.667,41.807,-82.066,170.046,35.808,156.741
C04230=1044.673,42.056,-82.083,170.047,35.810,156.741
C04231=1044.680,42.306,-82.100,170.049,35.811,156.741
C04232=1044.686,42.555,-82.117,170.051,35.813,156.741
C04233=1044.692,42.804,-82.133,170.052,35.814,156.742
C04234=1044.698,43.054,-82.151,170.054,35.815,156.742
C04235=1044.704,43.303,-82.167,170.056,35.816,156.742
C04236=1044.711,43.553,-82.185,170.058,35.818,156.742
C04237=1044.717,43.802,-82.201,170.059,35.819,156.742
C04238=1044.723,44.051,-82.218,170.062,35.821,156.743
C04239=1044.729,44.301,-82.235,170.064,35.822,156.743
C04240=1044.735,44.550,-82.252,170.065,35.823,156.743
C04241=1044.742,44.836,-82.271,170.067,35.825,156.744
C04242=1044.749,45.123,-82.292,170.069,35.827,156.744
C04243=1044.756,45.410,-82.311,170.071,35.829,156.744
C04244=1044.763,45.696,-82.330,170.073,35.830,156.744
C04245=1044.769,45.946,-82.347,170.076,35.832,156.745
C04246=1044.776,46.194,-82.364,170.077,35.833,156.745
C04247=1044.782,46.444,-82.381,170.079,35.834,156.745
C04248=1044.788,46.693,-82.399,170.081,35.836,156.745
C04249=1044.794,46.942,-82.416,170.082,35.837,156.746
C04250=1044.801,47.192,-82.432,170.084,35.839,156.746
C04251=1044.806,47.441,-82.450,170.086,35.840,156.746
C04252=1044.813,47.691,-82.467,170.087,35.841,156.746
C04253=1044.819,47.940,-82.483,170.089,35.843,156.747
C04254=1044.825,48.190,-82.501,170.092,35.844,156.747
C04255=1044.831,48.439,-82.518,170.093,35.846,156.747
C04256=1044.838,48.689,-82.535,170.095,35.847,156.747
C04257=1044.843,48.938,-82.552,170.097,35.848,156.748
C04258=1044.850,49.186,-82.569,170.098,35.850,156.748
C04259=1044.856,49.436,-82.587,170.100,35.851,156.748
C04260=1044.862,49.685,-82.604,170.102,35.853,156.749
C04261=1044.868,49.935,-82.621,170.103,35.854,156.749
C04262=1044.874,50.184,-82.639,170.106,35.856,156.749
C04263=1044.881,50.434,-82.655,170.108,35.857,156.749
C04264=1044.887,50.683,-82.672,170.110,35.858,156.749
C04265=1044.893,50.932,-82.690,170.111,35.860,156.750
C04266=1044.899,51.181,-82.707,170.113,35.861,156.750
C04267=1044.906,51.431,-82.724,170.115,35.863,156.750
C04268=1044.911,51.680,-82.741,170.116,35.864,156.750
C04269=1044.918,51.930,-82.759,170.118,35.865,156.751
C04270=1044.924,52.178,-82.776,170.121,35.867,156.751
C04271=1044.930,52.428,-82.793,170.122,35.868,156.751
C04272=1044.937,52.677,-82.810,170.124,35.870,156.751
C04273=1044.943,52.927,-82.827,170.126,35.871,156.752
C04274=1044.949,53.176,-82.845,170.127,35.872,156.752
C04275=1044.956,53.425,-82.862,170.129,35.873,156.752
C04276=1044.962,53.675,-82.880,170.131,35.875,156.753
C04277=1044.968,53.924,-82.897,170.132,35.877,156.753
C04278=1044.975,54.173,-82.914,170.135,35.878,156.753
C04279=1044.980,54.422,-82.932,170.137,35.879,156.753
C04280=1044.987,54.672,-82.948,170.138,35.880,156.753
C04281=1044.993,54.921,-82.965,170.140,35.882,156.754
C04282=1044.999,55.171,-82.983,170.142,35.884,156.754
C04283=1045.006,55.420,-83.001,170.143,35.885,156.754
C04284=1045.012,55.669,-83.018,170.145,35.886,156.754
C04285=1045.019,55.919,-83.036,170.147,35.888,156.755
C04286=1045.025,56.167,-83.053,170.149,35.889,156.755
C04287=1045.031,56.417,-83.070,170.151,35.890,156.755
C04288=1045.037,56.666,-83.087,170.153,35.892,156.755
C04289=1045.043,56.916,-83.105,170.154,35.893,156.756
C04290=1045.050,57.165,-83.123,170.156,35.895,156.756
C04291=1045.056,57.414,-83.140,170.158,35.896,156.756
C04292=1045.063,57.664,-83.158,170.160,35.897,156.756
C04293=1045.069,57.913,-83.175,170.161,35.898,156.757
C04294=1045.075,58.162,-83.193,170.163,35.900,156.757
C04295=1045.082,58.412,-83.210,170.166,35.902,156.757
C04296=1045.089,58.661,-83.227,170.167,35.903,156.757
C04297=1045.098,59.024,-83.252,170.170,35.905,156.758
C04298=1045.107,59.387,-83.278,170.172,35.907,156.758
C04299=1045.116,59.749,-83.304,170.175,35.909,156.758
C04300=1045.125,60.112,-83.329,170.177,35.911,156.759
C04301=1045.136,60.535,-83.359,170.181,35.913,156.759
C04302=1045.146,60.956,-83.388,170.184,35.915,156.760
C04303=1045.158,61.378,-83.417,170.187,35.918,156.760
C04304=1045.169,61.800,-83.447,170.189,35.920,156.761
C04305=1045.174,62.049,-83.465,170.191,35.921,156.761
C04306=1045.181,62.299,-83.482,170.194,35.923,156.761
C04307=1045.187,62.549,-83.500,170.196,35.924,156.761
C04308=1045.194,62.797,-83.518,170.197,35.925,156.761
C04309=1045.200,63.046,-83.536,170.199,35.926,156.762
C04310=1045.207,63.296,-83.553,170.201,35.928,156.762
C04311=1045.213,63.545,-83.570,170.202,35.929,156.762
C04312=1045.219,63.794,-83.588,170.204,35.930,156.762
C04313=1045.226,64.044,-83.605,170.206,35.932,156.763
C04314=1045.232,64.293,-83.623,170.208,35.933,156.763
C04315=1045.238,64.543,-83.642,170.210,35.935,156.763
C04316=1045.244,64.792,-83.659,170.212,35.936,156.763
C04317=1045.251,65.041,-83.677,170.213,35.938,156.764
C04318=1045.257,65.291,-83.695,170.215,35.939,156.764
C04319=1045.263,65.539,-83.713,170.217,35.941,156.764
C04320=1045.270,65.789,-83.730,170.218,35.942,156.764
C04321=1045.276,66.038,-83.748,170.220,35.944,156.765
C04322=1045.282,66.288,-83.766,170.223,35.945,156.765
C04323=1045.288,66.536,-83.784,170.224,35.946,156.765
C04324=1045.295,66.786,-83.802,170.226,35.948,156.765
C04325=1045.301,67.036,-83.820,170.228,35.949,156.766
C04326=1045.306,67.284,-83.838,170.229,35.951,156.766
C04327=1045.313,67.534,-83.855,170.231,35.952,156.766
C04328=1045.319,67.783,-83.873,170.233,35.953,156.766
C04329=1045.326,68.032,-83.892,170.234,35.955,156.767
C04330=1045.331,68.281,-83.909,170.237,35.956,156.767
C04331=1045.338,68.531,-83.927,170.239,35.958,156.767
C04332=1045.345,68.780,-83.945,170.240,35.959,156.768
C04333=1045.351,69.030,-83.963,170.242,35.961,156.768
C04334=1045.356,69.279,-83.981,170.244,35.962,156.768
C04335=1045.363,69.528,-83.999,170.245,35.963,156.768
C04336=1045.370,69.777,-84.017,170.247,35.965,156.769
C04337=1045.376,70.027,-84.036,170.250,35.967,156.769
C04338=1045.382,70.276,-84.053,170.251,35.968,156.769
C04339=1045.388,70.525,-84.071,170.253,35.969,156.769
C04340=1045.394,70.774,-84.090,170.254,35.971,156.770
C04341=1045.400,71.024,-84.108,170.256,35.972,156.770
C04342=1045.407,71.273,-84.126,170.258,35.974,156.770
C04343=1045.413,71.522,-84.143,170.259,35.975,156.771
C04344=1045.419,71.771,-84.162,170.261,35.977,156.771
C04345=1045.425,72.021,-84.180,170.264,35.978,156.771
C04346=1045.432,72.270,-84.198,170.265,35.979,156.771
C04347=1045.437,72.519,-84.216,170.267,35.981,156.772
C04348=1045.444,72.768,-84.235,170.269,35.982,156.772
C04349=1045.450,73.018,-84.253,170.270,35.984,156.772
C04350=1045.456,73.267,-84.271,170.272,35.986,156.772
C04351=1045.462,73.517,-84.289,170.274,35.987,156.773
C04352=1045.468,73.765,-84.307,170.276,35.988,156.773
C04353=1045.474,74.015,-84.325,170.278,35.990,156.773
C04354=1045.481,74.264,-84.344,170.280,35.991,156.773
C04355=1045.488,74.513,-84.361,170.281,35.993,156.774
C04356=1045.494,74.763,-84.380,170.283,35.995,156.774
C04357=1045.500,75.012,-84.398,170.285,35.996,156.774
C04358=1045.506,75.261,-84.416,170.286,35.997,156.774
C04359=1045.512,75.510,-84.435,170.288,35.998,156.775
C04360=1045.519,75.760,-84.453,170.291,36.000,156.775
C04361=1045.525,76.009,-84.471,170.292,36.001,156.775
C04362=1045.531,76.258,-84.489,170.294,36.003,156.775
C04363=1045.538,76.508,-84.508,170.296,36.005,156.776
C04364=1045.544,76.757,-84.527,170.297,36.006,156.776
C04365=1045.551,77.043,-84.547,170.299,36.007,156.776
C04366=1045.558,77.329,-84.568,170.302,36.009,156.777
C04367=1045.565,77.615,-84.590,170.304,36.011,156.777
C04368=1045.573,77.901,-84.611,170.306,36.012,156.777
C04369=1045.579,78.150,-84.629,170.307,36.014,156.778
C04370=1045.585,78.399,-84.647,170.309,36.015,156.778
C04371=1045.591,78.648,-84.665,170.311,36.017,156.778
C04372=1045.597,78.897,-84.685,170.312,36.019,156.778
C04373=1045.603,79.147,-84.703,170.315,36.020,156.779
C04374=1045.609,79.396,-84.721,170.317,36.022,156.779
C04375=1045.616,79.645,-84.740,170.318,36.023,156.779
C04376=1045.622,79.894,-84.759,170.320,36.024,156.779
C04377=1045.628,80.144,-84.776,170.322,36.026,156.780
C04378=1045.633,80.393,-84.795,170.323,36.027,156.780
C04379=1045.640,80.642,-84.814,170.325,36.029,156.780
C04380=1045.646,80.891,-84.833,170.328,36.031,156.781
C04381=1045.652,81.140,-84.851,170.329,36.032,156.781
C04382=1045.659,81.390,-84.869,170.331,36.034,156.781
C04383=1045.664,81.639,-84.888,170.332,36.035,156.781
C04384=1045.671,81.889,-84.907,170.334,36.037,156.782
C04385=1045.677,82.138,-84.926,170.336,36.038,156.782
C04386=1045.684,82.387,-84.944,170.337,36.039,156.782
C04387=1045.689,82.636,-84.962,170.340,36.041,156.783
C04388=1045.695,82.885,-84.981,170.342,36.043,156.783
C04389=1045.701,83.134,-85.000,170.343,36.044,156.783
C04390=1045.708,83.384,-85.019,170.345,36.046,156.783
C04391=1045.714,83.633,-85.037,170.347,36.047,156.784
C04392=1045.720,83.882,-85.056,170.348,36.049,156.784
C04393=1045.726,84.131,-85.075,170.350,36.050,156.784
C04394=1045.733,84.380,-85.094,170.353,36.051,156.784
C04395=1045.739,84.630,-85.112,170.354,36.053,156.785
C04396=1045.745,84.879,-85.130,170.356,36.055,156.785
C04397=1045.751,85.129,-85.150,170.358,36.056,156.785
C04398=1045.757,85.378,-85.168,170.359,36.058,156.786
C04399=1045.764,85.627,-85.187,170.361,36.059,156.786
C04400=1045.770,85.876,-85.205,170.363,36.060,156.786
C04401=1045.776,86.125,-85.225,170.365,36.062,156.786
C04402=1045.782,86.375,-85.243,170.367,36.063,156.787
C04403=1045.789,86.624,-85.262,170.369,36.065,156.787
C04404=1045.795,86.873,-85.281,170.370,36.067,156.787
C04405=1045.801,87.122,-85.300,170.372,36.068,156.787
C04406=1045.807,87.371,-85.319,170.374,36.070,156.788
C04407=1045.814,87.620,-85.337,170.375,36.071,156.788
C04408=1045.820,87.870,-85.356,170.378,36.072,156.788
C04409=1045.826,88.119,-85.375,170.380,36.074,156.789
C04410=1045.832,88.368,-85.394,170.381,36.075,156.789
C04411=1045.839,88.617,-85.412,170.383,36.077,156.789
C04412=1045.845,88.866,-85.431,170.385,36.079,156.789
C04413=1045.851,89.116,-85.450,170.386,36.080,156.790
C04414=1045.857,89.365,-85.469,170.388,36.081,156.790
C04415=1045.864,89.614,-85.488,170.391,36.083,156.790
C04416=1045.870,89.863,-85.506,170.392,36.084,156.791
C04417=1045.876,90.113,-85.525,170.394,36.086,156.791
C04418=1045.882,90.362,-85.544,170.396,36.087,156.791
C04419=1045.888,90.611,-85.563,170.397,36.089,156.791
C04420=1045.894,90.860,-85.582,170.399,36.090,156.792
C04421=1045.901,91.109,-85.601,170.401,36.092,156.792
C04422=1045.907,91.358,-85.621,170.403,36.093,156.792
C04423=1045.913,91.607,-85.639,170.405,36.095,156.792
C04424=1045.919,91.857,-85.659,170.406,36.096,156.793
C04425=1045.925,92.106,-85.677,170.408,36.098,156.793
C04426=1045.931,92.356,-85.697,170.410,36.099,156.793
C04427=1045.937,92.605,-85.717,170.411,36.101,156.794
C04428=1045.944,92.854,-85.735,170.414,36.103,156.794
C04429=1045.950,93.140,-85.757,170.416,36.104,156.794
C04430=1045.958,93.425,-85.779,170.418,36.106,156.795
C04431=1045.965,93.712,-85.801,170.420,36.108,156.795
C04432=1045.972,93.998,-85.824,170.422,36.109,156.795
C04433=1045.978,94.247,-85.842,170.423,36.111,156.796
C04434=1045.984,94.496,-85.861,170.426,36.113,156.796
C04435=1045.990,94.745,-85.880,170.428,36.115,156.796
C04436=1045.996,94.994,-85.900,170.429,36.116,156.796
C04437=1046.003,95.243,-85.919,170.431,36.118,156.797
C04438=1046.008,95.493,-85.938,170.433,36.119,156.797
C04439=1046.015,95.741,-85.957,170.434,36.120,156.797
C04440=1046.021,95.991,-85.977,170.436,36.122,156.798
C04441=1046.028,96.240,-85.996,170.439,36.123,156.798
C04442=1046.033,96.490,-86.015,170.440,36.125,156.798
C04443=1046.040,96.738,-86.034,170.442,36.126,156.798
C04444=1046.046,96.988,-86.053,170.444,36.128,156.799
C04445=1046.052,97.237,-86.073,170.445,36.130,156.799
C04446=1046.058,97.486,-86.092,170.447,36.131,156.799
C04447=1046.064,97.735,-86.111,170.450,36.133,156.800
C04448=1046.070,97.984,-86.130,170.451,36.134,156.800
C04449=1046.077,98.234,-86.150,170.453,36.136,156.800
C04450=1046.083,98.483,-86.169,170.455,36.137,156.800
C04451=1046.089,98.732,-86.189,170.456,36.138,156.801
C04452=1046.096,98.981,-86.208,170.458,36.140,156.801
C04453=1046.101,99.230,-86.227,170.460,36.142,156.801
C04454=1046.107,99.479,-86.247,170.462,36.143,156.802
C04455=1046.115,99.729,-86.266,170.464,36.145,156.802
C04456=1046.121,99.978,-86.286,170.466,36.146,156.802
C04457=1046.127,100.227,-86.304,170.468,36.148,156.802
C04458=1046.133,100.476,-86.324,170.469,36.149,156.803
C04459=1046.139,100.725,-86.344,170.471,36.151,156.803
C04460=1046.145,100.974,-86.362,170.473,36.152,156.803
C04461=1046.152,101.224,-86.383,170.475,36.154,156.804
C04462=1046.157,101.473,-86.402,170.477,36.155,156.804
C04463=1046.163,101.722,-86.422,170.479,36.157,156.804
C04464=1046.169,101.971,-86.441,170.480,36.159,156.804
C04465=1046.176,102.220,-86.460,170.482,36.160,156.805
C04466=1046.181,102.469,-86.480,170.484,36.162,156.805
C04467=1046.188,102.719,-86.500,170.486,36.164,156.805
C04468=1046.194,102.968,-86.520,170.488,36.165,156.806
C04469=1046.200,103.217,-86.539,170.490,36.167,156.806
C04470=1046.206,103.466,-86.559,170.491,36.169,156.806
C04471=1046.212,103.715,-86.578,170.493,36.170,156.806
C04472=1046.218,103.964,-86.598,170.495,36.172,156.807
C04473=1046.224,104.214,-86.617,170.497,36.173,156.807
C04474=1046.230,104.463,-86.637,170.499,36.175,156.807
C04475=1046.236,104.712,-86.657,170.501,36.176,156.808
C04476=1046.242,104.961,-86.676,170.502,36.178,156.808
C04477=1046.249,105.210,-86.696,170.504,36.179,156.808
C04478=1046.255,105.460,-86.715,170.506,36.181,156.809
C04479=1046.261,105.709,-86.735,170.508,36.182,156.809
C04480=1046.267,105.957,-86.755,170.510,36.184,156.809
C04481=1046.273,106.207,-86.775,170.512,36.185,156.809
C04482=1046.279,106.456,-86.795,170.513,36.187,156.810
C04483=1046.286,106.705,-86.814,170.515,36.189,156.810
C04484=1046.292,106.954,-86.834,170.517,36.190,156.810
C04485=1046.298,107.203,-86.853,170.519,36.192,156.811
C04486=1046.304,107.453,-86.874,170.521,36.194,156.811
C04487=1046.310,107.702,-86.893,170.523,36.195,156.811
C04488=1046.316,107.951,-86.913,170.525,36.197,156.812
C04489=1046.323,108.200,-86.933,170.526,36.198,156.812
C04490=1046.329,108.449,-86.953,170.528,36.199,156.812
C04491=1046.335,108.698,-86.972,170.530,36.201,156.812
C04492=1046.341,108.947,-86.992,170.532,36.202,156.813
C04493=1046.348,109.233,-87.015,170.534,36.204,156.813
C04494=1046.356,109.519,-87.038,170.536,36.206,156.813
C04495=1046.363,109.805,-87.060,170.538,36.208,156.814
C04496=1046.370,110.091,-87.083,170.540,36.210,156.814
C04497=1046.376,110.340,-87.103,170.543,36.211,156.814
C04498=1046.382,110.589,-87.123,170.545,36.213,156.815
C04499=1046.389,110.838,-87.143,170.546,36.214,156.815
C04500=1046.395,111.087,-87.163,170.548,36.216,156.815
C04501=1046.400,111.337,-87.182,170.550,36.217,156.815
C04502=1046.407,111.586,-87.203,170.551,36.219,156.816
C04503=1046.413,111.835,-87.223,170.553,36.221,156.816
C04504=1046.419,112.084,-87.243,170.556,36.222,156.816
C04505=1046.425,112.333,-87.263,170.557,36.224,156.817
C04506=1046.431,112.582,-87.283,170.559,36.226,156.817
C04507=1046.437,112.831,-87.303,170.561,36.227,156.817
C04508=1046.444,113.081,-87.322,170.563,36.229,156.818
C04509=1046.450,113.330,-87.342,170.565,36.231,156.818
C04510=1046.456,113.579,-87.362,170.567,36.232,156.818
C04511=1046.462,113.828,-87.383,170.569,36.234,156.818
C04512=1046.468,114.077,-87.403,170.570,36.235,156.819
C04513=1046.474,114.326,-87.423,170.572,36.237,156.819
C04514=1046.480,114.576,-87.443,170.574,36.239,156.819
C04515=1046.486,114.824,-87.463,170.576,36.240,156.820
C04516=1046.492,115.073,-87.483,170.578,36.242,156.820
C04517=1046.497,115.322,-87.504,170.580,36.244,156.820
C04518=1046.504,115.572,-87.524,170.581,36.245,156.821
C04519=1046.510,115.821,-87.544,170.583,36.247,156.821
C04520=1046.515,116.070,-87.565,170.585,36.249,156.821
C04521=1046.522,116.319,-87.585,170.588,36.250,156.822
C04522=1046.528,116.568,-87.605,170.589,36.252,156.822
C04523=1046.534,116.817,-87.625,170.591,36.254,156.822
C04524=1046.540,117.067,-87.646,170.593,36.255,156.823
C04525=1046.546,117.315,-87.667,170.594,36.257,156.823
C04526=1046.552,117.564,-87.687,170.596,36.259,156.823
C04527=1046.558,117.814,-87.707,170.599,36.260,156.823
C04528=1046.564,118.062,-87.727,170.600,36.262,156.824
C04529=1046.570,118.312,-87.748,170.602,36.264,156.824
C04530=1046.576,118.561,-87.768,170.604,36.265,156.824
C04531=1046.582,118.810,-87.788,170.606,36.267,156.825
C04532=1046.588,119.059,-87.809,170.608,36.269,156.825
C04533=1046.594,119.308,-87.829,170.610,36.270,156.825
C04534=1046.600,119.557,-87.850,170.612,36.272,156.826
C04535=1046.606,119.806,-87.870,170.613,36.273,156.826
C04536=1046.612,120.055,-87.890,170.615,36.275,156.826
C04537=1046.618,120.305,-87.911,170.617,36.277,156.827
C04538=1046.624,120.554,-87.931,170.620,36.278,156.827
C04539=1046.631,120.803,-87.951,170.621,36.280,156.827
C04540=1046.637,121.051,-87.972,170.623,36.282,156.828
C04541=1046.642,121.300,-87.993,170.625,36.283,156.828
C04542=1046.649,121.550,-88.013,170.626,36.285,156.828
C04543=1046.655,121.799,-88.033,170.628,36.286,156.828
C04544=1046.661,122.048,-88.054,170.631,36.288,156.829
C04545=1046.667,122.297,-88.074,170.633,36.290,156.829
C04546=1046.674,122.546,-88.095,170.634,36.291,156.829
C04547=1046.679,122.795,-88.115,170.636,36.293,156.830
C04548=1046.686,123.044,-88.136,170.638,36.295,156.830
C04549=1046.692,123.293,-88.156,170.640,36.296,156.830
C04550=1046.698,123.543,-88.177,170.642,36.298,156.831
C04551=1046.704,123.792,-88.197,170.644,36.299,156.831
C04552=1046.711,124.041,-88.218,170.646,36.301,156.831
C04553=1046.716,124.290,-88.239,170.648,36.303,156.832
C04554=1046.722,124.539,-88.259,170.649,36.304,156.832
C04555=1046.729,124.788,-88.280,170.652,36.306,156.832
C04556=1046.735,125.037,-88.301,170.654,36.307,156.833
C04557=1046.742,125.323,-88.324,170.656,36.309,156.833
C04558=1046.748,125.609,-88.347,170.658,36.311,156.833
C04559=1046.755,125.894,-88.371,170.660,36.313,156.834
C04560=1046.763,126.180,-88.395,170.662,36.315,156.834
C04561=1046.769,126.429,-88.415,170.665,36.316,156.834
C04562=1046.775,126.678,-88.437,170.666,36.318,156.835
C04563=1046.781,126.927,-88.457,170.668,36.320,156.835
C04564=1046.788,127.177,-88.477,170.670,36.321,156.835
C04565=1046.793,127.425,-88.498,170.672,36.323,156.835
C04566=1046.800,127.675,-88.518,170.674,36.325,156.836
C04567=1046.807,127.924,-88.539,170.676,36.326,156.836
C04568=1046.812,128.173,-88.560,170.678,36.328,156.836
C04569=1046.819,128.422,-88.581,170.680,36.330,156.837
C04570=1046.824,128.671,-88.602,170.682,36.331,156.837
C04571=1046.831,128.920,-88.622,170.683,36.333,156.837
C04572=1046.838,129.169,-88.643,170.686,36.335,156.838
C04573=1046.843,129.418,-88.664,170.688,36.336,156.838
C04574=1046.850,129.667,-88.685,170.690,36.338,156.838
C04575=1046.856,129.916,-88.705,170.691,36.339,156.839
C04576=1046.862,130.165,-88.726,170.693,36.341,156.839
C04577=1046.869,130.415,-88.746,170.695,36.342,156.839
C04578=1046.874,130.663,-88.768,170.698,36.344,156.840
C04579=1046.881,130.913,-88.788,170.700,36.346,156.840
C04580=1046.887,131.161,-88.809,170.701,36.347,156.840
C04581=1046.893,131.411,-88.830,170.703,36.349,156.841
C04582=1046.900,131.660,-88.851,170.705,36.351,156.841
C04583=1046.905,131.908,-88.872,170.708,36.352,156.841
C04584=1046.911,132.158,-88.893,170.710,36.354,156.841
C04585=1046.917,132.406,-88.914,170.711,36.356,156.842
C04586=1046.923,132.656,-88.935,170.713,36.357,156.842
C04587=1046.930,132.905,-88.956,170.715,36.359,156.842
C04588=1046.936,133.153,-88.977,170.718,36.361,156.843
C04589=1046.942,133.403,-88.998,170.719,36.362,156.843
C04590=1046.947,133.652,-89.019,170.721,36.364,156.843
C04591=1046.954,133.901,-89.040,170.723,36.366,156.844
C04592=1046.960,134.150,-89.061,170.725,36.367,156.844
C04593=1046.966,134.399,-89.082,170.727,36.369,156.844
C04594=1046.972,134.648,-89.103,170.729,36.370,156.845
C04595=1046.978,134.898,-89.124,170.731,36.372,156.845
C04596=1046.984,135.146,-89.145,170.733,36.374,156.845
C04597=1046.990,135.395,-89.167,170.735,36.375,156.846
C04598=1046.997,135.644,-89.188,170.736,36.377,156.846
C04599=1047.002,135.893,-89.209,170.739,36.379,156.846
C04600=1047.008,136.143,-89.230,170.741,36.381,156.847
C04601=1047.015,136.391,-89.251,170.743,36.382,156.847
C04602=1047.021,136.640,-89.273,170.745,36.384,156.847
C04603=1047.027,136.890,-89.294,170.746,36.386,156.848
C04604=1047.034,137.139,-89.315,170.749,36.388,156.848
C04605=1047.039,137.387,-89.336,170.751,36.389,156.848
C04606=1047.045,137.636,-89.358,170.753,36.391,156.849
C04607=1047.051,137.886,-89.379,170.755,36.393,156.849
C04608=1047.057,138.134,-89.399,170.756,36.395,156.849
C04609=1047.064,138.384,-89.421,170.758,36.396,156.850
C04610=1047.070,138.633,-89.442,170.761,36.398,156.850
C04611=1047.075,138.881,-89.464,170.763,36.400,156.850
C04612=1047.082,139.130,-89.485,170.765,36.401,156.851
C04613=1047.088,139.379,-89.506,170.767,36.403,156.851
C04614=1047.094,139.629,-89.527,170.768,36.405,156.851
C04615=1047.100,139.878,-89.549,170.771,36.406,156.852
C04616=1047.106,140.127,-89.570,170.773,36.408,156.852
C04617=1047.112,140.376,-89.592,170.775,36.409,156.852
C04618=1047.118,140.625,-89.613,170.777,36.411,156.853
C04619=1047.124,140.874,-89.635,170.778,36.413,156.853
C04620=1047.130,141.123,-89.656,170.781,36.415,156.853
C04621=1047.137,141.408,-89.681,170.783,36.417,156.854
C04622=1047.144,141.694,-89.705,170.785,36.419,156.854
C04623=1047.151,141.979,-89.730,170.787,36.421,156.855
C04624=1047.158,142.265,-89.754,170.791,36.423,156.855
C04625=1047.164,142.514,-89.776,170.792,36.425,156.855
C04626=1047.170,142.763,-89.797,170.794,36.427,156.856
C04627=1047.176,143.012,-89.819,170.796,36.428,156.856
C04628=1047.182,143.261,-89.840,170.798,36.430,156.856
C04629=1047.188,143.510,-89.862,170.801,36.432,156.857
C04630=1047.194,143.759,-89.883,170.802,36.434,156.857
C04631=1047.201,144.008,-89.906,170.804,36.435,156.857
C04632=1047.206,144.256,-89.927,170.806,36.437,156.858
C04633=1047.212,144.506,-89.949,170.808,36.438,156.858
C04634=1047.219,144.755,-89.970,170.811,36.440,156.858
C04635=1047.225,145.004,-89.992,170.813,36.442,156.859
C04636=1047.231,145.253,-90.014,170.815,36.444,156.859
C04637=1047.236,145.502,-90.035,170.816,36.445,156.859
C04638=1047.243,145.751,-90.056,170.818,36.447,156.860
C04639=1047.249,146.000,-90.078,170.820,36.449,156.860
C04640=1047.255,146.249,-90.100,170.823,36.451,156.860
C04641=1047.261,146.498,-90.122,170.825,36.453,156.861
C04642=1047.267,146.746,-90.143,170.827,36.454,156.861
C04643=1047.274,146.995,-90.164,170.829,36.456,156.861
C04644=1047.280,147.244,-90.186,170.830,36.458,156.862
C04645=1047.285,147.494,-90.208,170.833,36.459,156.862
C04646=1047.292,147.743,-90.230,170.835,36.461,156.862
C04647=1047.298,147.992,-90.252,170.837,36.463,156.863
C04648=1047.304,148.240,-90.273,170.839,36.465,156.863
C04649=1047.310,148.489,-90.295,170.842,36.467,156.863
C04650=1047.316,148.739,-90.317,170.844,36.468,156.864
C04651=1047.322,148.987,-90.339,170.845,36.470,156.864
C04652=1047.329,149.236,-90.361,170.847,36.472,156.864
C04653=1047.334,149.486,-90.383,170.849,36.474,156.865
C04654=1047.340,149.734,-90.404,170.852,36.475,156.865
C04655=1047.346,149.983,-90.427,170.854,36.477,156.866
C04656=1047.352,150.232,-90.448,170.856,36.479,156.866
C04657=1047.358,150.481,-90.470,170.858,36.481,156.866
C04658=1047.365,150.730,-90.492,170.859,36.483,156.867
C04659=1047.370,150.980,-90.514,170.862,36.485,156.867
C04660=1047.376,151.229,-90.536,170.864,36.486,156.867
C04661=1047.382,151.477,-90.558,170.866,36.488,156.868
C04662=1047.388,151.726,-90.580,170.868,36.490,156.868
C04663=1047.394,151.975,-90.602,170.870,36.491,156.868
C04664=1047.400,152.224,-90.624,170.873,36.493,156.869
C04665=1047.407,152.473,-90.646,170.875,36.495,156.869
C04666=1047.413,152.722,-90.668,170.876,36.497,156.869
C04667=1047.419,152.971,-90.690,170.878,36.499,156.870
C04668=1047.425,153.221,-90.712,170.880,36.501,156.870
C04669=1047.431,153.469,-90.734,170.883,36.503,156.871
C04670=1047.437,153.718,-90.756,170.885,36.504,156.871
C04671=1047.443,153.966,-90.778,170.887,36.506,156.871
C04672=1047.448,154.216,-90.800,170.889,36.508,156.872
C04673=1047.455,154.464,-90.823,170.892,36.509,156.872
C04674=1047.461,154.713,-90.844,170.894,36.511,156.872
C04675=1047.468,154.962,-90.867,170.896,36.513,156.873
C04676=1047.473,155.212,-90.889,170.897,36.515,156.873
C04677=1047.479,155.460,-90.911,170.899,36.517,156.873
C04678=1047.485,155.710,-90.933,170.902,36.519,156.874
C04679=1047.491,155.958,-90.956,170.904,36.520,156.874
C04680=1047.498,156.207,-90.977,170.906,36.522,156.874
C04681=1047.503,156.456,-91.000,170.908,36.524,156.875
C04682=1047.509,156.706,-91.022,170.910,36.526,156.875
C04683=1047.516,156.954,-91.044,170.913,36.528,156.875
C04684=1047.522,157.203,-91.067,170.915,36.530,156.876
C04685=1047.528,157.488,-91.092,170.917,36.532,156.876
C04686=1047.535,157.774,-91.118,170.919,36.534,156.877
C04687=1047.542,158.058,-91.143,170.922,36.536,156.877
C04688=1047.549,158.344,-91.169,170.924,36.538,156.878
C04689=1047.555,158.593,-91.192,170.926,36.540,156.878
C04690=1047.561,158.842,-91.213,170.928,36.542,156.878
C04691=1047.568,159.091,-91.236,170.931,36.544,156.879
C04692=1047.574,159.340,-91.259,170.933,36.546,156.879
C04693=1047.580,159.589,-91.280,170.935,36.547,156.879
C04694=1047.585,159.838,-91.303,170.937,36.549,156.880
C04695=1047.592,160.086,-91.325,170.939,36.551,156.880
C04696=1047.598,160.335,-91.348,170.942,36.553,156.880
C04697=1047.604,160.585,-91.370,170.944,36.555,156.881
C04698=1047.610,160.833,-91.393,170.946,36.557,156.881
C04699=1047.616,161.082,-91.415,170.948,36.558,156.882
C04700=1047.622,161.331,-91.438,170.951,36.561,156.882
C04701=1047.627,161.580,-91.461,170.953,36.563,156.882
C04702=1047.633,161.829,-91.483,170.954,36.565,156.883
C04703=1047.639,162.078,-91.506,170.956,36.566,156.883
C04704=1047.645,162.327,-91.529,170.959,36.568,156.884
C04705=1047.651,162.576,-91.552,170.961,36.571,156.884
C04706=1047.657,162.825,-91.575,170.963,36.572,156.884
C04707=1047.662,163.074,-91.598,170.965,36.574,156.885
C04708=1047.668,163.323,-91.619,170.967,36.576,156.885
C04709=1047.674,163.572,-91.642,170.970,36.578,156.885
C04710=1047.680,163.821,-91.665,170.972,36.580,156.886
C04711=1047.686,164.069,-91.688,170.974,36.582,156.886
C04712=1047.691,164.318,-91.711,170.976,36.584,156.887
C04713=1047.698,164.567,-91.733,170.979,36.586,156.887
C04714=1047.704,164.816,-91.756,170.981,36.588,156.887
C04715=1047.709,165.065,-91.779,170.983,36.590,156.888
C04716=1047.715,165.314,-91.802,170.984,36.592,156.888
C04717=1047.721,165.562,-91.825,170.987,36.594,156.889
C04718=1047.727,165.811,-91.848,170.989,36.596,156.889
C04719=1047.733,166.060,-91.870,170.991,36.598,156.889
C04720=1047.739,166.309,-91.893,170.993,36.600,156.890
C04721=1047.744,166.558,-91.916,170.996,36.602,156.890
C04722=1047.750,166.807,-91.939,170.998,36.604,156.891
C04723=1047.757,167.055,-91.962,171.000,36.606,156.891
C04724=1047.762,167.304,-91.985,171.002,36.607,156.891
C04725=1047.768,167.553,-92.008,171.005,36.610,156.892
C04726=1047.774,167.803,-92.031,171.007,36.612,156.892
C04727=1047.780,168.052,-92.054,171.009,36.613,156.893
C04728=1047.787,168.300,-92.076,171.011,36.615,156.893
C04729=1047.792,168.549,-92.099,171.013,36.617,156.893
C04730=1047.798,168.798,-92.122,171.016,36.620,156.894
C04731=1047.804,169.047,-92.145,171.018,36.621,156.894
C04732=1047.810,169.296,-92.168,171.020,36.623,156.895
C04733=1047.816,169.544,-92.192,171.022,36.625,156.895
C04734=1047.823,169.793,-92.214,171.025,36.627,156.895
C04735=1047.828,170.042,-92.237,171.027,36.629,156.896
C04736=1047.834,170.291,-92.260,171.029,36.631,156.896
C04737=1047.840,170.540,-92.283,171.031,36.633,156.896
C04738=1047.846,170.789,-92.306,171.034,36.635,156.897
C04739=1047.852,171.037,-92.330,171.036,36.637,156.897
C04740=1047.859,171.286,-92.352,171.038,36.639,156.898
C04741=1047.864,171.535,-92.375,171.040,36.641,156.898
C04742=1047.870,171.784,-92.398,171.043,36.643,156.898
C04743=1047.876,172.033,-92.421,171.045,36.645,156.899
C04744=1047.882,172.281,-92.445,171.047,36.647,156.899
C04745=1047.888,172.531,-92.468,171.049,36.649,156.900
C04746=1047.894,172.780,-92.491,171.052,36.651,156.900
C04747=1047.900,173.028,-92.514,171.054,36.652,156.900
C04748=1047.906,173.277,-92.537,171.056,36.655,156.901
C04749=1047.913,173.562,-92.564,171.059,36.657,156.901
C04750=1047.920,173.847,-92.590,171.062,36.659,156.902
C04751=1047.927,174.132,-92.617,171.064,36.662,156.902
C04752=1047.934,174.417,-92.644,171.067,36.663,156.903
C04753=1047.940,174.666,-92.666,171.069,36.666,156.903
C04754=1047.946,174.914,-92.690,171.072,36.668,156.903
C04755=1047.952,175.163,-92.713,171.074,36.670,156.904
C04756=1047.958,175.412,-92.736,171.076,36.671,156.904
C04757=1047.965,175.661,-92.759,171.078,36.674,156.905
C04758=1047.970,175.910,-92.782,171.081,36.676,156.905
C04759=1047.977,176.159,-92.806,171.083,36.677,156.905
C04760=1047.983,176.407,-92.829,171.085,36.679,156.906
C04761=1047.989,176.656,-92.852,171.087,36.682,156.906
C04762=1047.995,176.904,-92.875,171.090,36.684,156.907
C04763=1048.001,177.154,-92.899,171.092,36.685,156.907
C04764=1048.007,177.403,-92.922,171.094,36.687,156.907
C04765=1048.013,177.651,-92.945,171.096,36.690,156.908
C04766=1048.020,177.901,-92.969,171.099,36.691,156.908
C04767=1048.026,178.149,-92.992,171.102,36.693,156.909
C04768=1048.032,178.399,-93.016,171.104,36.695,156.909
C04769=1048.038,178.647,-93.039,171.106,36.698,156.910
C04770=1048.044,178.896,-93.062,171.109,36.699,156.910
C04771=1048.050,179.145,-93.086,171.111,36.701,156.910
C04772=1048.057,179.393,-93.109,171.113,36.703,156.911
C04773=1048.063,179.642,-93.132,171.115,36.705,156.911
C04774=1048.069,179.891,-93.156,171.118,36.707,156.911
C04775=1048.075,180.139,-93.179,171.120,36.709,156.912
C04776=1048.082,180.389,-93.203,171.122,36.711,156.912
C04777=1048.088,180.637,-93.226,171.125,36.713,156.913
C04778=1048.093,180.886,-93.249,171.128,36.715,156.913
C04779=1048.100,181.135,-93.273,171.130,36.717,156.913
C04780=1048.106,181.383,-93.297,171.132,36.719,156.914
C04781=1048.112,181.633,-93.320,171.134,36.721,156.914
C04782=1048.118,181.881,-93.344,171.137,36.723,156.915
C04783=1048.125,182.131,-93.367,171.139,36.725,156.915
C04784=1048.131,182.379,-93.391,171.141,36.727,156.916
C04785=1048.137,182.627,-93.414,171.144,36.729,156.916
C04786=1048.144,182.877,-93.437,171.147,36.731,156.916
C04787=1048.150,183.125,-93.461,171.149,36.733,156.917
C04788=1048.156,183.374,-93.485,171.151,36.735,156.917
C04789=1048.162,183.623,-93.508,171.154,36.737,156.918
C04790=1048.169,183.872,-93.532,171.156,36.739,156.918
C04791=1048.174,184.120,-93.556,171.158,36.741,156.918
C04792=1048.180,184.370,-93.579,171.160,36.744,156.919
C04793=1048.186,184.619,-93.604,171.164,36.745,156.919
C04794=1048.192,184.867,-93.627,171.166,36.748,156.920
C04795=1048.198,185.116,-93.651,171.168,36.750,156.920
C04796=1048.204,185.364,-93.676,171.170,36.752,156.921
C04797=1048.210,185.613,-93.700,171.173,36.754,156.921
C04798=1048.215,185.863,-93.723,171.175,36.756,156.921
C04799=1048.221,186.111,-93.747,171.177,36.759,156.922
C04800=1048.227,186.360,-93.771,171.180,36.761,156.922
C04801=1048.233,186.609,-93.795,171.182,36.763,156.923
C04802=1048.239,186.858,-93.820,171.185,36.765,156.923
C04803=1048.245,187.106,-93.843,171.187,36.767,156.924
C04804=1048.251,187.355,-93.868,171.190,36.770,156.924
C04805=1048.257,187.604,-93.892,171.192,36.772,156.925
C04806=1048.263,187.852,-93.916,171.194,36.774,156.925
C04807=1048.269,188.101,-93.940,171.197,36.776,156.925
C04808=1048.274,188.350,-93.964,171.199,36.778,156.926
C04809=1048.281,188.599,-93.988,171.202,36.781,156.926
C04810=1048.286,188.847,-94.013,171.204,36.782,156.927
C04811=1048.293,189.096,-94.037,171.207,36.785,156.927
C04812=1048.298,189.345,-94.061,171.209,36.787,156.928
C04813=1048.305,189.630,-94.088,171.211,36.790,156.928
C04814=1048.312,189.913,-94.116,171.215,36.792,156.929
C04815=1048.319,190.198,-94.143,171.217,36.795,156.929
C04816=1048.326,190.483,-94.171,171.220,36.797,156.930
C04817=1048.332,190.732,-94.195,171.223,36.799,156.930
C04818=1048.339,190.980,-94.220,171.225,36.801,156.931
C04819=1048.344,191.229,-94.244,171.227,36.804,156.931
C04820=1048.350,191.477,-94.268,171.230,36.806,156.932
C04821=1048.356,191.726,-94.292,171.233,36.808,156.932
C04822=1048.362,191.975,-94.316,171.235,36.810,156.933
C04823=1048.368,192.224,-94.340,171.237,36.813,156.933
C04824=1048.374,192.473,-94.365,171.240,36.814,156.933
C04825=1048.380,192.721,-94.389,171.243,36.817,156.934
C04826=1048.386,192.970,-94.414,171.245,36.819,156.934
C04827=1048.392,193.219,-94.438,171.247,36.821,156.935
C04828=1048.398,193.467,-94.462,171.250,36.823,156.935
C04829=1048.404,193.716,-94.486,171.252,36.826,156.936
C04830=1048.410,193.965,-94.511,171.255,36.828,156.936
C04831=1048.417,194.213,-94.535,171.258,36.830,156.937
C04832=1048.423,194.463,-94.560,171.260,36.833,156.937
C04833=1048.429,194.711,-94.584,171.262,36.834,156.938
C04834=1048.434,194.960,-94.608,171.265,36.837,156.938
C04835=1048.441,195.208,-94.633,171.268,36.839,156.939
C04836=1048.447,195.457,-94.657,171.270,36.841,156.939
C04837=1048.453,195.706,-94.682,171.272,36.843,156.939
C04838=1048.459,195.955,-94.706,171.275,36.846,156.940
C04839=1048.465,196.203,-94.731,171.278,36.848,156.940
C04840=1048.472,196.452,-94.755,171.280,36.850,156.941
C04841=1048.477,196.701,-94.779,171.283,36.852,156.941
C04842=1048.484,196.949,-94.804,171.285,36.855,156.942
C04843=1048.490,197.199,-94.829,171.288,36.857,156.942
C04844=1048.495,197.447,-94.853,171.291,36.859,156.943
C04845=1048.502,197.696,-94.878,171.293,36.861,156.943
C04846=1048.508,197.945,-94.902,171.295,36.863,156.944
C04847=1048.514,198.194,-94.926,171.298,36.866,156.944
C04848=1048.520,198.442,-94.951,171.301,36.868,156.945
C04849=1048.527,198.691,-94.975,171.303,36.870,156.945
C04850=1048.533,198.939,-95.000,171.305,36.872,156.945
C04851=1048.538,199.188,-95.025,171.309,36.875,156.946
C04852=1048.545,199.436,-95.049,171.311,36.877,156.946
C04853=1048.551,199.686,-95.074,171.313,36.879,156.947
C04854=1048.558,199.935,-95.098,171.316,36.881,156.947
C04855=1048.564,200.183,-95.123,171.319,36.884,156.948
C04856=1048.569,200.432,-95.148,171.321,36.886,156.948
C04857=1048.576,200.680,-95.172,171.323,36.888,156.949
C04858=1048.582,200.930,-95.197,171.327,36.890,156.949
C04859=1048.589,201.178,-95.222,171.329,36.893,156.950
C04860=1048.595,201.426,-95.247,171.331,36.895,156.950
C04861=1048.600,201.675,-95.271,171.335,36.898,156.951
C04862=1048.607,201.924,-95.297,171.337,36.900,156.951
C04863=1048.613,202.173,-95.321,171.339,36.902,156.952
C04864=1048.618,202.421,-95.346,171.342,36.904,156.952
C04865=1048.624,202.670,-95.372,171.345,36.907,156.953
C04866=1048.631,202.919,-95.396,171.347,36.909,156.953
C04867=1048.637,203.167,-95.421,171.350,36.911,156.954
C04868=1048.643,203.416,-95.446,171.352,36.914,156.954
C04869=1048.649,203.665,-95.471,171.355,36.916,156.955
C04870=1048.655,203.913,-95.496,171.358,36.919,156.955
C04871=1048.661,204.162,-95.521,171.360,36.921,156.956
C04872=1048.667,204.411,-95.546,171.363,36.923,156.956
C04873=1048.673,204.659,-95.571,171.366,36.926,156.957
C04874=1048.679,204.908,-95.596,171.368,36.928,156.957
C04875=1048.685,205.157,-95.622,171.371,36.931,156.958
C04876=1048.691,205.406,-95.646,171.374,36.933,156.958
C04877=1048.717,206.458,-95.752,171.612,37.031,156.979
C04878=1048.724,206.719,-95.780,171.614,37.034,156.980
C04879=1048.731,206.980,-95.807,171.616,37.038,156.981
C04880=1048.738,207.241,-95.835,171.618,37.041,156.981
C04881=1048.744,207.502,-95.863,171.621,37.044,156.982
C04882=1048.751,207.750,-95.889,171.622,37.047,156.983
C04883=1048.758,207.999,-95.914,171.625,37.051,156.984
C04884=1048.763,208.248,-95.941,171.626,37.054,156.984
C04885=1048.770,208.496,-95.967,171.628,37.057,156.985
C04886=1048.777,208.744,-95.993,171.631,37.060,156.986
C04887=1048.783,208.992,-96.019,171.632,37.063,156.986
C04888=1048.790,209.242,-96.046,171.635,37.066,156.987
C04889=1048.796,209.490,-96.072,171.636,37.069,156.988
C04890=1048.803,209.739,-96.098,171.639,37.073,156.988
C04891=1048.809,209.987,-96.125,171.640,37.076,156.989
C04892=1048.815,210.235,-96.151,171.643,37.079,156.990
C04893=1048.822,210.484,-96.178,171.645,37.082,156.990
C04894=1048.828,210.732,-96.204,171.647,37.085,156.991
C04895=1048.835,210.982,-96.230,171.649,37.088,156.992
C04896=1048.841,211.230,-96.256,171.650,37.092,156.992
C04897=1048.848,211.479,-96.283,171.653,37.095,156.993
C04898=1048.855,211.727,-96.309,171.655,37.098,156.994
C04899=1048.861,211.976,-96.336,171.657,37.101,156.994
C04900=1048.867,212.224,-96.362,171.659,37.105,156.995
C04901=1048.873,212.472,-96.389,171.661,37.108,156.996
C04902=1048.880,212.721,-96.415,171.663,37.110,156.996
C04903=1048.886,212.970,-96.442,171.666,37.114,156.997
C04904=1048.892,213.219,-96.469,171.667,37.117,156.998
C04905=1048.899,213.467,-96.495,171.670,37.120,156.998
C04906=1048.905,213.716,-96.522,171.671,37.124,156.999
C04907=1048.912,213.964,-96.548,171.673,37.127,157.000
C04908=1048.918,214.213,-96.575,171.676,37.130,157.000
C04909=1048.925,214.461,-96.601,171.677,37.133,157.001
C04910=1048.931,214.709,-96.628,171.680,37.136,157.002
C04911=1048.938,214.957,-96.655,171.682,37.139,157.002
C04912=1048.944,215.206,-96.681,171.684,37.143,157.003
C04913=1048.950,215.455,-96.708,171.686,37.146,157.004
C04914=1048.957,215.703,-96.734,171.688,37.149,157.004
C04915=1048.963,215.952,-96.761,171.690,37.152,157.005
C04916=1048.970,216.200,-96.787,171.693,37.155,157.006
C04917=1048.976,216.449,-96.814,171.694,37.158,157.006
C04918=1048.983,216.697,-96.842,171.697,37.161,157.007
C04919=1048.989,216.945,-96.868,171.699,37.165,157.008
C04920=1048.995,217.195,-96.895,171.701,37.168,157.008
C04921=1049.002,217.443,-96.921,171.703,37.171,157.009
C04922=1049.008,217.692,-96.948,171.705,37.174,157.010
C04923=1049.015,217.939,-96.975,171.707,37.177,157.010
C04924=1049.022,218.188,-97.002,171.709,37.180,157.011
C04925=1049.028,218.436,-97.028,171.712,37.183,157.012
C04926=1049.034,218.685,-97.055,171.713,37.186,157.012
C04927=1049.041,218.934,-97.083,171.716,37.189,157.013
C04928=1049.048,219.182,-97.109,171.718,37.193,157.014
C04929=1049.054,219.431,-97.136,171.721,37.196,157.014
C04930=1049.061,219.679,-97.162,171.722,37.199,157.015
C04931=1049.067,219.927,-97.190,171.725,37.202,157.016
C04932=1049.074,220.176,-97.217,171.727,37.205,157.016
C04933=1049.080,220.424,-97.243,171.729,37.208,157.017
C04934=1049.087,220.691,-97.273,171.731,37.211,157.018
C04935=1049.094,220.958,-97.301,171.734,37.215,157.018
C04936=1049.101,221.224,-97.330,171.736,37.218,157.019
C04937=1049.107,221.491,-97.360,171.738,37.221,157.020
C04938=1049.114,221.740,-97.387,171.740,37.225,157.021
C04939=1049.120,221.988,-97.413,171.742,37.228,157.021
C04940=1049.127,222.236,-97.440,171.745,37.231,157.022
C04941=1049.133,222.485,-97.467,171.746,37.234,157.023
C04942=1049.139,222.733,-97.495,171.749,37.237,157.023
C04943=1049.146,222.982,-97.522,171.751,37.240,157.024
C04944=1049.152,223.230,-97.549,171.754,37.243,157.025
C04945=1049.158,223.479,-97.576,171.755,37.246,157.025
C04946=1049.166,223.727,-97.603,171.758,37.250,157.026
C04947=1049.171,223.975,-97.630,171.760,37.253,157.027
C04948=1049.178,224.224,-97.658,171.763,37.256,157.027
C04949=1049.184,224.473,-97.685,171.764,37.259,157.028
C04950=1049.191,224.720,-97.712,171.767,37.262,157.029
C04951=1049.197,224.970,-97.739,171.769,37.265,157.029
C04952=1049.204,225.218,-97.767,171.772,37.268,157.030
C04953=1049.210,225.466,-97.794,171.773,37.271,157.031
C04954=1049.217,225.714,-97.821,171.776,37.275,157.031
C04955=1049.223,225.963,-97.848,171.778,37.278,157.032
C04956=1049.229,226.211,-97.875,171.780,37.281,157.033
C04957=1049.236,226.460,-97.903,171.782,37.284,157.033
C04958=1049.243,226.708,-97.930,171.784,37.287,157.034
C04959=1049.249,226.957,-97.957,171.787,37.290,157.035
C04960=1049.255,227.205,-97.985,171.789,37.293,157.035
C04961=1049.261,227.454,-98.012,171.791,37.296,157.036
C04962=1049.269,227.702,-98.039,171.793,37.299,157.037
C04963=1049.276,227.951,-98.067,171.796,37.302,157.037
C04964=1049.282,228.198,-98.094,171.798,37.306,157.038
C04965=1049.288,228.447,-98.121,171.801,37.309,157.039
C04966=1049.295,228.696,-98.149,171.802,37.312,157.039
C04967=1049.301,228.944,-98.177,171.805,37.314,157.040
C04968=1049.307,229.193,-98.203,171.807,37.317,157.041
C04969=1049.314,229.441,-98.231,171.810,37.321,157.041
C04970=1049.320,229.690,-98.259,171.812,37.324,157.042
C04971=1049.327,229.938,-98.286,171.814,37.327,157.043
C04972=1049.332,230.186,-98.314,171.816,37.330,157.043
C04973=1049.339,230.435,-98.341,171.819,37.333,157.044
C04974=1049.346,230.684,-98.369,171.821,37.336,157.045
C04975=1049.352,230.932,-98.397,171.823,37.339,157.045
C04976=1049.358,231.180,-98.424,171.825,37.342,157.046
C04977=1049.365,231.428,-98.452,171.827,37.345,157.047
C04978=1049.372,231.677,-98.480,171.830,37.349,157.047
C04979=1049.378,231.925,-98.507,171.832,37.352,157.048
C04980=1049.385,232.173,-98.535,171.835,37.355,157.049
C04981=1049.390,232.422,-98.562,171.837,37.358,157.049
C04982=1049.397,232.671,-98.590,171.839,37.361,157.050
C04983=1049.403,232.919,-98.618,171.841,37.364,157.051
C04984=1049.410,233.167,-98.646,171.844,37.367,157.051
C04985=1049.416,233.416,-98.674,171.846,37.370,157.052
C04986=1049.422,233.664,-98.701,171.849,37.374,157.053
C04987=1049.429,233.912,-98.729,171.851,37.377,157.053
C04988=1049.436,234.161,-98.757,171.853,37.380,157.054
C04989=1049.441,234.410,-98.785,171.855,37.383,157.055
C04990=1049.448,234.668,-98.814,171.858,37.386,157.055
C04991=1049.455,234.927,-98.843,171.860,37.389,157.056
C04992=1049.462,235.186,-98.872,171.863,37.393,157.057
C04993=1049.468,235.446,-98.901,171.865,37.395,157.058
C04994=1049.475,235.693,-98.929,171.868,37.398,157.058
C04995=1049.481,235.942,-98.958,171.870,37.402,157.059
C04996=1049.488,236.191,-98.985,171.873,37.405,157.060
C04997=1049.495,236.439,-99.013,171.874,37.408,157.060
C04998=1049.500,236.687,-99.041,171.877,37.411,157.061
C04999=1049.507,236.936,-99.069,171.879,37.414,157.062
C05000=1049.513,237.184,-99.096,171.882,37.417,157.062
C05001=1049.520,237.432,-99.124,171.884,37.420,157.063
C05002=1049.526,237.681,-99.153,171.887,37.423,157.064
C05003=1049.533,237.929,-99.181,171.889,37.426,157.064
C05004=1049.540,238.177,-99.209,171.892,37.429,157.065
C05005=1049.546,238.426,-99.237,171.894,37.433,157.066
C05006=1049.552,238.675,-99.265,171.897,37.436,157.066
C05007=1049.559,238.922,-99.293,171.898,37.439,157.067
C05008=1049.565,239.171,-99.321,171.901,37.441,157.068
C05009=1049.571,239.419,-99.349,171.903,37.444,157.068
C05010=1049.578,239.667,-99.377,171.906,37.448,157.069
C05011=1049.584,239.916,-99.406,171.908,37.451,157.070
C05012=1049.591,240.164,-99.433,171.911,37.454,157.070
C05013=1049.598,240.412,-99.461,171.913,37.457,157.071
C05014=1049.604,240.661,-99.490,171.916,37.460,157.072
C05015=1049.611,240.909,-99.518,171.918,37.463,157.072
C05016=1049.617,241.158,-99.546,171.921,37.466,157.073
C05017=1049.624,241.406,-99.575,171.923,37.469,157.074
C05018=1049.630,241.654,-99.602,171.926,37.472,157.074
C05019=1049.636,241.903,-99.631,171.928,37.475,157.075
C05020=1049.642,242.151,-99.660,171.931,37.479,157.076
C05021=1049.649,242.399,-99.687,171.932,37.482,157.076
C05022=1049.655,242.647,-99.716,171.935,37.484,157.077
C05023=1049.662,242.896,-99.744,171.937,37.487,157.078
C05024=1049.668,243.144,-99.773,171.940,37.491,157.078
C05025=1049.674,243.393,-99.802,171.942,37.494,157.079
C05026=1049.681,243.641,-99.830,171.945,37.497,157.080
C05027=1049.687,243.889,-99.858,171.947,37.500,157.081
C05028=1049.694,244.137,-99.887,171.950,37.503,157.081
C05029=1049.700,244.386,-99.915,171.952,37.506,157.082
C05030=1049.706,244.634,-99.944,171.955,37.509,157.083
C05031=1049.713,244.883,-99.972,171.957,37.513,157.083
C05032=1049.719,245.131,-100.001,171.960,37.516,157.084
C05033=1049.726,245.379,-100.029,171.962,37.519,157.085
C05034=1049.732,245.627,-100.058,171.965,37.521,157.085
C05035=1049.738,245.875,-100.087,171.967,37.524,157.086
C05036=1049.744,246.124,-100.115,171.970,37.528,157.087
C05037=1049.751,246.372,-100.143,171.972,37.531,157.087
C05038=1049.758,246.620,-100.173,171.975,37.534,157.088
C05039=1049.764,246.869,-100.201,171.977,37.537,157.089
C05040=1049.770,247.117,-100.230,171.980,37.540,157.089
C05041=1049.776,247.365,-100.259,171.982,37.544,157.090
C05042=1049.782,247.614,-100.287,171.985,37.547,157.091
C05043=1049.789,247.862,-100.316,171.987,37.550,157.091
C05044=1049.795,248.110,-100.345,171.990,37.553,157.092
C05045=1049.801,248.358,-100.374,171.992,37.556,157.093
C05046=1049.808,248.611,-100.403,171.995,37.559,157.094
C05047=1049.814,248.865,-100.433,171.997,37.563,157.094
C05048=1049.821,249.118,-100.462,172.000,37.565,157.095
C05049=1049.827,249.372,-100.491,172.002,37.569,157.096
C05050=1049.833,249.620,-100.520,172.005,37.572,157.096
C05051=1049.840,249.868,-100.549,172.007,37.575,157.097
C05052=1049.846,250.116,-100.579,172.010,37.578,157.098
C05053=1049.853,250.364,-100.607,172.012,37.581,157.099
C05054=1049.859,250.613,-100.635,172.015,37.584,157.099
C05055=1049.865,250.861,-100.664,172.017,37.587,157.100
C05056=1049.872,251.109,-100.694,172.020,37.591,157.101
C05057=1049.878,251.358,-100.723,172.022,37.594,157.101
C05058=1049.884,251.606,-100.752,172.025,37.596,157.102
C05059=1049.891,251.854,-100.781,172.028,37.600,157.103
C05060=1049.897,252.102,-100.810,172.030,37.603,157.103
C05061=1049.903,252.350,-100.839,172.033,37.606,157.104
C05062=1049.910,252.598,-100.867,172.036,37.609,157.105
C05063=1049.917,252.847,-100.897,172.039,37.612,157.105
C05064=1049.923,253.095,-100.926,172.041,37.615,157.106
C05065=1049.930,253.343,-100.955,172.044,37.618,157.107
C05066=1049.936,253.591,-100.984,172.046,37.621,157.107
C05067=1049.942,253.839,-101.013,172.049,37.625,157.108
C05068=1049.949,254.088,-101.042,172.051,37.627,157.109
C05069=1049.955,254.336,-101.071,172.054,37.630,157.109
C05070=1049.961,254.584,-101.100,172.056,37.634,157.110
C05071=1049.968,254.833,-101.129,172.059,37.637,157.111
C05072=1049.974,255.081,-101.159,172.061,37.640,157.112
C05073=1049.981,255.329,-101.187,172.064,37.643,157.112
C05074=1049.988,255.577,-101.216,172.067,37.646,157.113
C05075=1049.994,255.825,-101.245,172.070,37.649,157.114
C05076=1050.000,256.074,-101.274,172.072,37.652,157.114
C05077=1050.007,256.322,-101.305,172.075,37.655,157.115
C05078=1050.014,256.570,-101.334,172.077,37.658,157.116
C05079=1050.020,256.818,-101.363,172.080,37.661,157.116
C05080=1050.027,257.067,-101.392,172.082,37.664,157.117
C05081=1050.033,257.315,-101.421,172.085,37.667,157.118
C05082=1050.039,257.563,-101.450,172.088,37.671,157.119
C05083=1050.046,257.811,-101.480,172.091,37.673,157.119
C05084=1050.053,258.060,-101.509,172.093,37.676,157.120
C05085=1050.059,258.308,-101.538,172.096,37.679,157.120
C05086=1050.065,258.556,-101.567,172.098,37.682,157.121
C05087=1050.072,258.804,-101.597,172.101,37.686,157.122
C05088=1050.079,259.052,-101.627,172.105,37.689,157.123
C05089=1050.085,259.300,-101.656,172.107,37.692,157.123
C05090=1050.092,259.549,-101.685,172.110,37.694,157.124
C05091=1050.098,259.797,-101.715,172.112,37.698,157.125
C05092=1050.106,260.045,-101.744,172.115,37.701,157.125
C05093=1050.112,260.293,-101.773,172.117,37.704,157.126
C05094=1050.119,260.541,-101.802,172.121,37.707,157.127
C05095=1050.125,260.790,-101.832,172.123,37.710,157.127
C05096=1050.132,261.038,-101.861,172.126,37.713,157.128
C05097=1050.139,261.286,-101.891,172.128,37.716,157.129
C05098=1050.145,261.534,-101.920,172.131,37.719,157.129
C05099=1050.152,261.782,-101.950,172.134,37.722,157.130
C05100=1050.159,262.030,-101.979,172.137,37.725,157.131
C05101=1050.165,262.278,-102.009,172.139,37.728,157.132
C05102=1050.171,262.530,-102.039,172.142,37.731,157.132
C05103=1050.178,262.781,-102.069,172.144,37.734,157.133
C05104=1050.184,263.033,-102.099,172.148,37.737,157.134
C05105=1050.191,263.285,-102.129,172.151,37.740,157.134
C05106=1050.198,263.533,-102.159,172.153,37.744,157.135
C05107=1050.204,263.781,-102.188,172.156,37.747,157.136
C05108=1050.211,264.030,-102.219,172.159,37.750,157.137
C05109=1050.217,264.278,-102.248,172.162,37.753,157.137
C05110=1050.223,264.525,-102.278,172.164,37.756,157.138
C05111=1050.230,264.774,-102.308,172.167,37.759,157.139
C05112=1050.236,265.022,-102.337,172.169,37.762,157.139
C05113=1050.243,265.270,-102.368,172.173,37.765,157.140
C05114=1050.249,265.518,-102.398,172.176,37.769,157.141
C05115=1050.255,265.767,-102.428,172.178,37.772,157.141
C05116=1050.262,266.015,-102.457,172.181,37.775,157.142
C05117=1050.268,266.262,-102.487,172.184,37.778,157.143
C05118=1050.275,266.511,-102.517,172.187,37.781,157.144
C05119=1050.281,266.759,-102.547,172.189,37.784,157.144
C05120=1050.288,267.007,-102.577,172.192,37.787,157.145
C05121=1050.294,267.255,-102.607,172.194,37.790,157.146
C05122=1050.301,267.504,-102.637,172.198,37.794,157.146
C05123=1050.308,267.751,-102.667,172.200,37.797,157.147
C05124=1050.314,268.000,-102.697,172.203,37.799,157.148
C05125=1050.320,268.247,-102.727,172.207,37.803,157.149
C05126=1050.327,268.496,-102.758,172.209,37.806,157.149
C05127=1050.333,268.743,-102.787,172.212,37.809,157.150
C05128=1050.340,268.992,-102.817,172.214,37.812,157.151
C05129=1050.346,269.240,-102.847,172.218,37.816,157.152
C05130=1050.353,269.488,-102.878,172.220,37.819,157.152
C05131=1050.359,269.736,-102.908,172.223,37.821,157.153
C05132=1050.366,269.984,-102.938,172.225,37.825,157.154
C05133=1050.372,270.232,-102.968,172.229,37.828,157.154
C05134=1050.378,270.480,-102.999,172.232,37.831,157.155
C05135=1050.385,270.728,-103.029,172.234,37.834,157.156
C05136=1050.391,270.976,-103.059,172.238,37.837,157.156
C05137=1050.399,271.225,-103.089,172.240,37.840,157.157
C05138=1050.404,271.472,-103.120,172.243,37.843,157.158
C05139=1050.412,271.721,-103.150,172.246,37.847,157.159
C05140=1050.417,271.968,-103.180,172.249,37.850,157.159
C05141=1050.425,272.217,-103.210,172.252,37.853,157.160
C05142=1050.430,272.464,-103.241,172.254,37.856,157.161
C05143=1050.437,272.713,-103.271,172.258,37.860,157.162
C05144=1050.444,272.961,-103.302,172.260,37.862,157.162
C05145=1050.450,273.209,-103.332,172.263,37.866,157.163
C05146=1050.456,273.458,-103.363,172.266,37.869,157.164
C05147=1050.463,273.704,-103.393,172.269,37.872,157.165
C05148=1050.469,273.953,-103.424,172.272,37.875,157.165
C05149=1050.475,274.201,-103.454,172.275,37.879,157.166
C05150=1050.482,274.449,-103.484,172.278,37.881,157.167
C05151=1050.489,274.698,-103.515,172.280,37.885,157.167
C05152=1050.495,274.945,-103.546,172.284,37.888,157.168
C05153=1050.502,275.193,-103.576,172.286,37.891,157.169
C05154=1050.509,275.441,-103.607,172.289,37.894,157.170
C05155=1050.514,275.689,-103.637,172.293,37.898,157.170
C05156=1050.521,275.937,-103.669,172.295,37.900,157.171
C05157=1050.528,276.186,-103.699,172.298,37.904,157.172
C05158=1050.534,276.441,-103.730,172.301,37.907,157.173
C05159=1050.541,276.697,-103.762,172.304,37.910,157.173
C05160=1050.547,276.953,-103.794,172.308,37.914,157.174
C05161=1050.555,277.209,-103.825,172.310,37.917,157.175
C05162=1050.561,277.457,-103.856,172.314,37.920,157.176
C05163=1050.567,277.705,-103.887,172.316,37.923,157.176
C05164=1050.574,277.953,-103.918,172.319,37.926,157.177
C05165=1050.580,278.201,-103.948,172.323,37.930,157.178
C05166=1050.587,278.449,-103.979,172.325,37.933,157.179
C05167=1050.594,278.697,-104.010,172.329,37.936,157.179
C05168=1050.599,278.945,-104.041,172.331,37.939,157.180
C05169=1050.606,279.193,-104.072,172.334,37.942,157.181
C05170=1050.613,279.441,-104.102,172.337,37.945,157.181
C05171=1050.620,279.689,-104.134,172.340,37.949,157.182
C05172=1050.626,279.937,-104.164,172.344,37.952,157.183
C05173=1050.633,280.185,-104.196,172.346,37.955,157.184
C05174=1050.639,280.433,-104.226,172.349,37.959,157.185
C05175=1050.646,280.681,-104.258,172.352,37.961,157.185
C05176=1050.652,280.928,-104.289,172.355,37.965,157.186
C05177=1050.658,281.177,-104.319,172.359,37.968,157.187
C05178=1050.665,281.425,-104.351,172.361,37.971,157.187
C05179=1050.671,281.672,-104.381,172.364,37.975,157.188
C05180=1050.678,281.920,-104.413,172.367,37.978,157.189
C05181=1050.684,282.168,-104.444,172.370,37.981,157.190
C05182=1050.691,282.417,-104.475,172.374,37.984,157.191
C05183=1050.697,282.665,-104.506,172.376,37.988,157.191
C05184=1050.704,282.912,-104.537,172.380,37.991,157.192
C05185=1050.710,283.160,-104.568,172.382,37.994,157.193
C05186=1050.717,283.408,-104.599,172.386,37.997,157.194
C05187=1050.723,283.657,-104.631,172.389,38.000,157.194
C05188=1050.729,283.904,-104.663,172.391,38.004,157.195
C05189=1050.735,284.152,-104.693,172.395,38.007,157.196
C05190=1050.742,284.400,-104.725,172.397,38.010,157.197
C05191=1050.749,284.648,-104.756,172.401,38.014,157.197
C05192=1050.755,284.896,-104.788,172.404,38.016,157.198
C05193=1050.762,285.144,-104.819,172.407,38.020,157.199
C05194=1050.769,285.392,-104.850,172.410,38.023,157.200
C05195=1050.775,285.640,-104.881,172.413,38.026,157.200
C05196=1050.781,285.887,-104.912,172.416,38.030,157.201
C05197=1050.788,286.135,-104.944,172.420,38.033,157.202
C05198=1050.795,286.383,-104.975,172.422,38.036,157.203
C05199=1050.802,286.631,-105.007,172.426,38.039,157.203
C05200=1050.808,286.879,-105.038,172.429,38.043,157.204
C05201=1050.815,287.127,-105.069,172.432,38.045,157.205
C05202=1050.822,287.375,-105.101,172.435,38.049,157.206
C05203=1050.828,287.623,-105.132,172.438,38.052,157.207
C05204=1050.834,287.871,-105.164,172.441,38.055,157.207
C05205=1050.841,288.119,-105.196,172.445,38.059,157.208
C05206=1050.848,288.367,-105.227,172.447,38.062,157.209
C05207=1050.854,288.614,-105.258,172.451,38.065,157.210
C05208=1050.860,288.862,-105.290,172.455,38.069,157.210
C05209=1050.867,289.110,-105.322,172.457,38.072,157.211
C05210=1050.873,289.358,-105.353,172.461,38.075,157.212
C05211=1050.880,289.606,-105.385,172.463,38.079,157.213
C05212=1050.886,289.854,-105.417,172.467,38.082,157.214
C05213=1050.893,290.101,-105.449,172.470,38.085,157.214
C05214=1050.900,290.369,-105.482,172.473,38.089,157.215
C05215=1050.907,290.636,-105.516,172.477,38.092,157.216
C05216=1050.915,290.904,-105.550,172.480,38.096,157.217
C05217=1050.921,291.171,-105.585,172.484,38.100,157.218
C05218=1050.928,291.419,-105.616,172.487,38.103,157.218
C05219=1050.934,291.666,-105.649,172.490,38.106,157.219
C05220=1050.941,291.914,-105.681,172.493,38.109,157.220
C05221=1050.948,292.162,-105.712,172.496,38.113,157.221
C05222=1050.954,292.410,-105.745,172.500,38.116,157.222
C05223=1050.961,292.658,-105.776,172.503,38.120,157.222
C05224=1050.967,292.906,-105.808,172.506,38.122,157.223
C05225=1050.974,293.153,-105.840,172.510,38.126,157.224
C05226=1050.980,293.401,-105.872,172.512,38.129,157.225
C05227=1050.986,293.649,-105.904,172.516,38.133,157.226
C05228=1050.994,293.897,-105.936,172.520,38.136,157.226
C05229=1051.001,294.145,-105.968,172.522,38.140,157.227
C05230=1051.007,294.393,-106.000,172.526,38.143,157.228
C05231=1051.014,294.641,-106.032,172.528,38.146,157.229
C05232=1051.020,294.889,-106.064,172.532,38.149,157.230
C05233=1051.027,295.136,-106.096,172.536,38.153,157.230
C05234=1051.033,295.384,-106.128,172.538,38.156,157.231
C05235=1051.040,295.632,-106.160,172.542,38.159,157.232
C05236=1051.046,295.880,-106.192,172.546,38.163,157.233
C05237=1051.053,296.127,-106.224,172.548,38.166,157.234
C05238=1051.059,296.375,-106.256,172.552,38.170,157.234
C05239=1051.065,296.623,-106.289,172.555,38.173,157.235
C05240=1051.072,296.870,-106.321,172.558,38.176,157.236
C05241=1051.079,297.119,-106.354,172.562,38.180,157.237
C05242=1051.085,297.367,-106.387,172.565,38.183,157.238
C05243=1051.091,297.614,-106.419,172.568,38.187,157.238
C05244=1051.097,297.863,-106.451,172.572,38.191,157.239
C05245=1051.104,298.110,-106.483,172.575,38.194,157.240
C05246=1051.111,298.357,-106.516,172.579,38.197,157.241
C05247=1051.117,298.605,-106.549,172.581,38.201,157.242
C05248=1051.123,298.853,-106.581,172.585,38.204,157.243
C05249=1051.130,299.101,-106.613,172.589,38.208,157.243
C05250=1051.136,299.348,-106.646,172.591,38.211,157.244
C05251=1051.143,299.596,-106.679,172.595,38.214,157.245
C05252=1051.149,299.844,-106.712,172.599,38.218,157.246
C05253=1051.155,300.092,-106.744,172.601,38.222,157.247
C05254=1051.162,300.340,-106.776,172.605,38.225,157.248
C05255=1051.169,300.587,-106.809,172.609,38.229,157.249
C05256=1051.175,300.835,-106.841,172.611,38.232,157.249
C05257=1051.182,301.083,-106.874,172.615,38.235,157.250
C05258=1051.188,301.331,-106.907,172.619,38.239,157.251
C05259=1051.195,301.578,-106.940,172.622,38.242,157.252
C05260=1051.202,301.825,-106.972,172.625,38.246,157.253
C05261=1051.208,302.073,-107.005,172.629,38.250,157.254
C05262=1051.215,302.321,-107.038,172.633,38.253,157.254
C05263=1051.221,302.569,-107.071,172.635,38.256,157.255
C05264=1051.227,302.817,-107.103,172.639,38.260,157.256
C05265=1051.234,303.064,-107.136,172.643,38.263,157.257
C05266=1051.241,303.312,-107.169,172.645,38.267,157.258
C05267=1051.248,303.560,-107.201,172.649,38.270,157.259
C05268=1051.254,303.807,-107.234,172.653,38.274,157.259
C05269=1051.261,304.056,-107.267,172.657,38.277,157.260
C05270=1051.268,304.338,-107.304,172.660,38.281,157.261
C05271=1051.276,304.621,-107.342,172.664,38.285,157.262
C05272=1051.283,304.905,-107.380,172.668,38.289,157.263
C05273=1051.291,305.188,-107.418,172.672,38.293,157.264
C05274=1051.297,305.436,-107.451,172.676,38.297,157.265
C05275=1051.304,305.684,-107.483,172.679,38.300,157.266
C05276=1051.311,305.931,-107.516,172.683,38.304,157.267
C05277=1051.318,306.180,-107.549,172.686,38.307,157.268
C05278=1051.324,306.427,-107.582,172.689,38.311,157.268
C05279=1051.331,306.674,-107.615,172.693,38.314,157.269
C05280=1051.337,306.922,-107.648,172.697,38.318,157.270
C05281=1051.344,307.170,-107.681,172.700,38.321,157.271
C05282=1051.351,307.418,-107.715,172.703,38.325,157.272
C05283=1051.357,307.665,-107.747,172.707,38.329,157.273
C05284=1051.364,307.913,-107.779,172.711,38.332,157.274
C05285=1051.371,308.160,-107.813,172.714,38.335,157.274
C05286=1051.378,308.408,-107.846,172.718,38.339,157.275
C05287=1051.385,308.656,-107.879,172.721,38.343,157.276
C05288=1051.391,308.903,-107.913,172.725,38.346,157.277
C05289=1051.398,309.151,-107.946,172.728,38.349,157.278
C05290=1051.405,309.398,-107.979,172.732,38.353,157.279
C05291=1051.412,309.647,-108.012,172.736,38.357,157.280
C05292=1051.418,309.894,-108.045,172.739,38.360,157.280
C05293=1051.425,310.142,-108.079,172.743,38.364,157.281
C05294=1051.431,310.390,-108.112,172.746,38.367,157.282
C05295=1051.439,310.637,-108.145,172.750,38.371,157.283
C05296=1051.446,310.885,-108.178,172.753,38.374,157.284
C05297=1051.453,311.132,-108.211,172.757,38.378,157.285
C05298=1051.460,311.381,-108.244,172.761,38.381,157.286
C05299=1051.466,311.627,-108.278,172.765,38.385,157.286
C05300=1051.473,311.876,-108.311,172.768,38.389,157.287
C05301=1051.480,312.123,-108.344,172.772,38.392,157.288
C05302=1051.487,312.370,-108.378,172.775,38.396,157.289
C05303=1051.494,312.619,-108.411,172.779,38.399,157.290
C05304=1051.500,312.866,-108.445,172.782,38.403,157.291
C05305=1051.507,313.114,-108.478,172.786,38.407,157.292
C05306=1051.513,313.361,-108.512,172.790,38.410,157.293
C05307=1051.520,313.609,-108.546,172.794,38.414,157.294
C05308=1051.527,313.856,-108.579,172.797,38.418,157.295
C05309=1051.533,314.105,-108.613,172.801,38.421,157.295
C05310=1051.540,314.351,-108.646,172.804,38.425,157.296
C05311=1051.546,314.599,-108.681,172.808,38.428,157.297
C05312=1051.553,314.847,-108.715,172.812,38.432,157.298
C05313=1051.559,315.094,-108.749,172.815,38.436,157.299
C05314=1051.567,315.342,-108.783,172.819,38.440,157.300
C05315=1051.572,315.589,-108.817,172.823,38.444,157.301
C05316=1051.580,315.837,-108.850,172.827,38.447,157.302
C05317=1051.585,316.084,-108.885,172.831,38.451,157.303
C05318=1051.593,316.332,-108.918,172.834,38.455,157.304
C05319=1051.599,316.580,-108.953,172.837,38.459,157.305
C05320=1051.606,316.827,-108.986,172.841,38.463,157.306
C05321=1051.612,317.075,-109.021,172.845,38.466,157.306
C05322=1051.619,317.323,-109.054,172.848,38.470,157.307
C05323=1051.625,317.570,-109.089,172.852,38.474,157.308
C05324=1051.632,317.818,-109.122,172.856,38.478,157.309
C05325=1051.639,318.066,-109.157,172.860,38.481,157.310
C05326=1051.646,318.354,-109.196,172.864,38.486,157.311
C05327=1051.654,318.640,-109.235,172.869,38.490,157.312
C05328=1051.661,318.928,-109.275,172.873,38.495,157.313
C05329=1051.669,319.216,-109.315,172.878,38.499,157.315
C05330=1051.676,319.463,-109.349,172.881,38.503,157.316
C05331=1051.683,319.711,-109.384,172.885,38.506,157.316
C05332=1051.690,319.959,-109.417,172.889,38.510,157.317
C05333=1051.696,320.206,-109.451,172.893,38.514,157.318
C05334=1051.704,320.453,-109.486,172.897,38.518,157.319
C05335=1051.710,320.701,-109.520,172.900,38.522,157.320
C05336=1051.717,320.949,-109.554,172.904,38.525,157.321
C05337=1051.723,321.196,-109.588,172.908,38.529,157.322
C05338=1051.730,321.444,-109.623,172.912,38.533,157.323
C05339=1051.737,321.691,-109.657,172.916,38.537,157.324
C05340=1051.743,321.939,-109.692,172.920,38.541,157.325
C05341=1051.751,322.186,-109.726,172.923,38.545,157.326
C05342=1051.757,322.434,-109.761,172.927,38.549,157.327
C05343=1051.764,322.682,-109.795,172.931,38.552,157.328
C05344=1051.771,322.929,-109.829,172.935,38.556,157.329
C05345=1051.777,323.177,-109.864,172.939,38.560,157.330
C05346=1051.785,323.424,-109.898,172.943,38.564,157.331
C05347=1051.791,323.672,-109.933,172.946,38.568,157.332
C05348=1051.798,323.920,-109.966,172.950,38.571,157.333
C05349=1051.805,324.167,-110.002,172.954,38.575,157.334
C05350=1051.812,324.415,-110.036,172.958,38.579,157.335
C05351=1051.819,324.662,-110.070,172.962,38.583,157.336
C05352=1051.826,324.910,-110.105,172.966,38.587,157.337
C05353=1051.832,325.157,-110.140,172.969,38.591,157.338
C05354=1051.840,325.405,-110.174,172.973,38.595,157.338
C05355=1051.846,325.652,-110.209,172.977,38.599,157.339
C05356=1051.854,325.899,-110.244,172.981,38.603,157.340
C05357=1051.860,326.147,-110.278,172.985,38.606,157.341
C05358=1051.867,326.395,-110.313,172.990,38.610,157.342
C05359=1051.874,326.642,-110.347,172.994,38.614,157.343
C05360=1051.881,326.890,-110.382,172.997,38.618,157.344
C05361=1051.888,327.137,-110.417,173.001,38.622,157.345
C05362=1051.895,327.385,-110.451,173.005,38.626,157.346
C05363=1051.902,327.632,-110.486,173.009,38.630,157.347
C05364=1051.909,327.879,-110.521,173.013,38.634,157.348
C05365=1051.916,328.127,-110.556,173.017,38.638,157.349
C05366=1051.923,328.375,-110.590,173.022,38.641,157.350
C05367=1051.930,328.622,-110.625,173.025,38.645,157.351
C05368=1051.937,328.870,-110.660,173.029,38.649,157.352
C05369=1051.944,329.117,-110.695,173.033,38.653,157.353
C05370=1051.952,329.364,-110.730,173.037,38.657,157.354
C05371=1051.958,329.612,-110.764,173.041,38.661,157.355
C05372=1051.965,329.859,-110.800,173.046,38.665,157.356
C05373=1051.972,330.107,-110.835,173.050,38.669,157.357
C05374=1051.978,330.354,-110.870,173.054,38.673,157.358
C05375=1051.985,330.602,-110.905,173.057,38.677,157.359
C05376=1051.993,330.850,-110.940,173.061,38.681,157.360
C05377=1051.999,331.097,-110.976,173.065,38.685,157.361
C05378=1052.006,331.344,-111.011,173.069,38.689,157.362
C05379=1052.013,331.592,-111.046,173.074,38.693,157.363
C05380=1052.020,331.839,-111.081,173.078,38.697,157.364
C05381=1052.027,332.086,-111.117,173.082,38.702,157.365
C05382=1052.034,332.369,-111.158,173.087,38.706,157.367
C05383=1052.042,332.651,-111.198,173.091,38.711,157.368
C05384=1052.051,332.933,-111.238,173.096,38.716,157.369
C05385=1052.058,333.216,-111.278,173.100,38.720,157.370
C05386=1052.065,333.464,-111.314,173.105,38.724,157.371
C05387=1052.072,333.711,-111.349,173.109,38.728,157.372
C05388=1052.079,333.959,-111.384,173.113,38.733,157.373
C05389=1052.086,334.205,-111.420,173.117,38.737,157.374
C05390=1052.093,334.453,-111.455,173.122,38.741,157.375
C05391=1052.100,334.701,-111.491,173.126,38.745,157.376
C05392=1052.107,334.948,-111.526,173.130,38.749,157.378
C05393=1052.114,335.195,-111.562,173.134,38.753,157.379
C05394=1052.121,335.443,-111.597,173.139,38.757,157.380
C05395=1052.127,335.691,-111.633,173.142,38.761,157.381
C05396=1052.134,335.937,-111.669,173.146,38.766,157.382
C05397=1052.141,336.185,-111.704,173.150,38.770,157.383
C05398=1052.149,336.432,-111.740,173.155,38.774,157.384
C05399=1052.155,336.680,-111.775,173.159,38.778,157.385
C05400=1052.162,336.927,-111.812,173.163,38.782,157.386
C05401=1052.169,337.175,-111.847,173.167,38.787,157.387
C05402=1052.176,337.421,-111.883,173.172,38.791,157.388
C05403=1052.183,337.669,-111.918,173.176,38.795,157.389
C05404=1052.190,337.917,-111.955,173.180,38.799,157.390
C05405=1052.197,338.163,-111.991,173.184,38.804,157.391
C05406=1052.204,338.411,-112.026,173.189,38.808,157.393
C05407=1052.211,338.658,-112.063,173.193,38.812,157.394
C05408=1052.217,338.906,-112.098,173.197,38.816,157.395
C05409=1052.225,339.153,-112.134,173.202,38.821,157.396
C05410=1052.231,339.400,-112.170,173.206,38.825,157.397
C05411=1052.238,339.647,-112.206,173.210,38.830,157.398
C05412=1052.245,339.895,-112.242,173.215,38.833,157.399
C05413=1052.252,340.142,-112.278,173.219,38.838,157.400
C05414=1052.260,340.390,-112.314,173.223,38.842,157.401
C05415=1052.266,340.637,-112.351,173.228,38.847,157.402
C05416=1052.274,340.885,-112.386,173.232,38.851,157.404
C05417=1052.281,341.131,-112.422,173.236,38.855,157.405
C05418=1052.288,341.379,-112.459,173.241,38.860,157.406
